LIN {X 0,Y 573.904,Z 122.065,A -85,B 0,C 180,E1 -2263.779,E2 -2263.779} C_VEL
LIN {X 0,Y 573.412,Z 118.44,A -85,B 0,C 180,E1 -2263.85,E2 -2263.85} C_VEL
LIN {X 0,Y 573.598,Z 96.264,A -85,B 0,C 180,E1 -2266.868,E2 -2266.868} C_VEL
LIN {X 0,Y 573.791,Z 74.375,A -85,B 0,C 180,E1 -2269.851,E2 -2269.851} C_VEL
LIN {X 0,Y 573.97,Z 52.577,A -85,B 0,C 180,E1 -2272.877,E2 -2272.877} C_VEL
LIN {X 0,Y 573.666,Z 48.09,A -85,B 0,C 180,E1 -2273.521,E2 -2273.521} C_VEL
LIN {X 0,Y 573.275,Z 46.079,A -85,B 0,C 180,E1 -2273.823,E2 -2273.823} C_VEL
LIN {X 0,Y 573.237,Z 46.08,A -85,B 0,C 180,E1 -2276.492,E2 -2276.492} C_VEL
LIN {X 0,Y 573.237,Z 46.078,A -85,B 0,C 180,E1 -2278.564,E2 -2278.564} C_VEL
LIN {X 0,Y 573.23,Z 46.075,A -85,B 0,C 180,E1 -2280.993,E2 -2280.993} C_VEL
LIN {X 0,Y 573.264,Z 46.076,A -85,B 0,C 180,E1 -2283.524,E2 -2283.524} C_VEL
LIN {X 0,Y 573.216,Z 46.083,A -85,B 0,C 180,E1 -2286.051,E2 -2286.051} C_VEL
LIN {X 0,Y 573.25,Z 46.073,A -85,B 0,C 180,E1 -2288.701,E2 -2288.701} C_VEL
LIN {X 0,Y 573.23,Z 46.085,A -85,B 0,C 180,E1 -2291.593,E2 -2291.593} C_VEL
LIN {X 0,Y 573.222,Z 46.077,A -85,B 0,C 180,E1 -2294.335,E2 -2294.335} C_VEL
LIN {X 0,Y 573.241,Z 46.083,A -85,B 0,C 180,E1 -2297.358,E2 -2297.358} C_VEL
LIN {X 0,Y 573.238,Z 46.075,A -85,B 0,C 180,E1 -2300.392,E2 -2300.392} C_VEL
LIN {X 0,Y 573.252,Z 46.08,A -85,B 0,C 180,E1 -2303.077,E2 -2303.077} C_VEL
LIN {X 0,Y 573.269,Z 46.073,A -85,B 0,C 180,E1 -2305.671,E2 -2305.671} C_VEL
LIN {X 0,Y 573.245,Z 46.074,A -85,B 0,C 180,E1 -2308.185,E2 -2308.185} C_VEL
LIN {X 0,Y 573.26,Z 46.076,A -85,B 0,C 180,E1 -2310.634,E2 -2310.634} C_VEL
LIN {X 0,Y 573.251,Z 46.081,A -85,B 0,C 180,E1 -2313.024,E2 -2313.024} C_VEL
LIN {X 0,Y 573.274,Z 46.073,A -85,B 0,C 180,E1 -2315.366,E2 -2315.366} C_VEL
LIN {X 0,Y 573.227,Z 46.08,A -85,B 0,C 180,E1 -2318.419,E2 -2318.419} C_VEL
LIN {X 0,Y 573.269,Z 46.08,A -85,B 0,C 180,E1 -2320.731,E2 -2320.731} C_VEL
LIN {X 0,Y 573.241,Z 46.074,A -85,B 0,C 180,E1 -2323.621,E2 -2323.621} C_VEL
LIN {X 0,Y 573.226,Z 46.086,A -85,B 0,C 180,E1 -2326.529,E2 -2326.529} C_VEL
LIN {X 0,Y 573.263,Z 46.076,A -85,B 0,C 180,E1 -2328.745,E2 -2328.745} C_VEL
LIN {X 0,Y 573.281,Z 46.069,A -85,B 0,C 180,E1 -2331.541,E2 -2331.541} C_VEL
LIN {X 0,Y 573.246,Z 46.075,A -85,B 0,C 180,E1 -2333.665,E2 -2333.665} C_VEL
LIN {X 0,Y 573.229,Z 46.079,A -85,B 0,C 180,E1 -2335.782,E2 -2335.782} C_VEL
LIN {X 0,Y 573.312,Z 46.071,A -85,B 0,C 180,E1 -2337.893,E2 -2337.893} C_VEL
LIN {X 0,Y 573.32,Z 46.066,A -85,B 0,C 180,E1 -2340.703,E2 -2340.703} C_VEL
LIN {X 0,Y 573.294,Z 46.068,A -85,B 0,C 180,E1 -2342.811,E2 -2342.811} C_VEL
LIN {X 0,Y 573.29,Z 46.073,A -85,B 0,C 180,E1 -2345.628,E2 -2345.628} C_VEL
LIN {X 0,Y 573.253,Z 46.074,A -85,B 0,C 180,E1 -2348.46,E2 -2348.46} C_VEL
LIN {X 0,Y 573.273,Z 46.074,A -85,B 0,C 180,E1 -2351.312,E2 -2351.312} C_VEL
LIN {X 0,Y 573.263,Z 46.072,A -85,B 0,C 180,E1 -2354.417,E2 -2354.417} C_VEL
LIN {X 0,Y 573.249,Z 46.076,A -85,B 0,C 180,E1 -2357.112,E2 -2357.112} C_VEL
LIN {X 0,Y 573.237,Z 46.076,A -85,B 0,C 180,E1 -2360.077,E2 -2360.077} C_VEL
LIN {X 0,Y 573.224,Z 46.076,A -85,B 0,C 180,E1 -2362.339,E2 -2362.339} C_VEL
LIN {X 0,Y 573.201,Z 46.079,A -85,B 0,C 180,E1 -2364.361,E2 -2364.361} C_VEL
LIN {X 0,Y 572.564,Z 46.164,A -85,B 0,C 180,E1 -2364.947,E2 -2364.947} C_VEL
LIN {X 0,Y 569.745,Z 46.52,A -85,B 0,C 180,E1 -2365.899,E2 -2365.899} C_VEL
LIN {X 0,Y 567.34,Z 46.822,A -85,B 0,C 180,E1 -2366.665,E2 -2366.665} C_VEL
LIN {X 0,Y 566.291,Z 46.949,A -85,B 0,C 180,E1 -2367.257,E2 -2367.257} C_VEL
LIN {X 0,Y 566.198,Z 46.957,A -85,B 0,C 180,E1 -2367.457,E2 -2367.457} C_VEL
LIN {X 0,Y 566.196,Z 46.953,A -85,B 0,C 180,E1 -2369.77,E2 -2369.77} C_VEL
LIN {X 0,Y 566.202,Z 46.952,A -85,B 0,C 180,E1 -2372.43,E2 -2372.43} C_VEL
LIN {X 0,Y 566.179,Z 46.964,A -85,B 0,C 180,E1 -2374.989,E2 -2374.989} C_VEL
LIN {X 0,Y 566.196,Z 46.954,A -85,B 0,C 180,E1 -2377.461,E2 -2377.461} C_VEL
LIN {X 0,Y 566.207,Z 46.952,A -85,B 0,C 180,E1 -2380.2,E2 -2380.2} C_VEL
LIN {X 0,Y 566.189,Z 46.957,A -85,B 0,C 180,E1 -2383.056,E2 -2383.056} C_VEL
LIN {X 0,Y 566.194,Z 46.954,A -85,B 0,C 180,E1 -2386.05,E2 -2386.05} C_VEL
LIN {X 0,Y 566.204,Z 46.952,A -85,B 0,C 180,E1 -2389.215,E2 -2389.215} C_VEL
LIN {X 0,Y 566.178,Z 46.954,A -85,B 0,C 180,E1 -2391.636,E2 -2391.636} C_VEL
LIN {X 0,Y 566.145,Z 46.967,A -85,B 0,C 180,E1 -2394.307,E2 -2394.307} C_VEL
LIN {X 0,Y 566.212,Z 46.951,A -85,B 0,C 180,E1 -2396.898,E2 -2396.898} C_VEL
LIN {X 0,Y 566.18,Z 46.954,A -85,B 0,C 180,E1 -2399.407,E2 -2399.407} C_VEL
LIN {X 0,Y 566.191,Z 46.958,A -85,B 0,C 180,E1 -2401.856,E2 -2401.856} C_VEL
LIN {X 0,Y 566.188,Z 46.959,A -85,B 0,C 180,E1 -2404.25,E2 -2404.25} C_VEL
LIN {X 0,Y 566.17,Z 46.956,A -85,B 0,C 180,E1 -2406.72,E2 -2406.72} C_VEL
LIN {X 0,Y 566.207,Z 46.956,A -85,B 0,C 180,E1 -2409.663,E2 -2409.663} C_VEL
LIN {X 0,Y 566.175,Z 46.964,A -85,B 0,C 180,E1 -2411.921,E2 -2411.921} C_VEL
LIN {X 0,Y 566.194,Z 46.954,A -85,B 0,C 180,E1 -2414.891,E2 -2414.891} C_VEL
LIN {X 0,Y 566.233,Z 46.954,A -85,B 0,C 180,E1 -2418.183,E2 -2418.183} C_VEL
LIN {X 0,Y 566.243,Z 47.146,A -85,B 0,C 180,E1 -2418.546,E2 -2418.546} C_VEL
LIN {X 0,Y 566.429,Z 52.827,A -85,B 0,C 180,E1 -2419.636,E2 -2419.636} C_VEL
LIN {X 0,Y 566.254,Z 68.023,A -85,B 0,C 180,E1 -2422.512,E2 -2422.512} C_VEL
LIN {X 0,Y 566.247,Z 70.905,A -85,B 0,C 180,E1 -2423.058,E2 -2423.058} C_VEL
LIN {X 0,Y 567.171,Z 77.845,A -85,B 0,C 180,E1 -2423.171,E2 -2423.171} C_VEL
LIN {X 0,Y 566.914,Z 176.791,A -85,B 0,C 180,E1 -2424.442,E2 -2424.442} C_VEL
LIN {X 0,Y 566.831,Z 189.95,A -85,B 0,C 180,E1 -2424.754,E2 -2424.754} C_VEL
LIN {X 0,Y 566.741,Z 202.54,A -85,B 0,C 180,E1 -2425.199,E2 -2425.199} C_VEL
LIN {X 0,Y 566.658,Z 213.764,A -85,B 0,C 180,E1 -2425.733,E2 -2425.733} C_VEL
LIN {X 0,Y 566.475,Z 225.38,A -85,B 0,C 180,E1 -2426.444,E2 -2426.444} C_VEL
LIN {X 0,Y 566.328,Z 235.815,A -85,B 0,C 180,E1 -2427.244,E2 -2427.244} C_VEL
LIN {X 0,Y 566.197,Z 246.089,A -85,B 0,C 180,E1 -2428.222,E2 -2428.222} C_VEL
LIN {X 0,Y 566.095,Z 255.035,A -85,B 0,C 180,E1 -2429.289,E2 -2429.289} C_VEL
LIN {X 0,Y 566.04,Z 262.266,A -85,B 0,C 180,E1 -2430.356,E2 -2430.356} C_VEL
LIN {X 0,Y 565.903,Z 268.085,A -85,B 0,C 180,E1 -2431.423,E2 -2431.423} C_VEL
LIN {X 0,Y 565.951,Z 272.675,A -85,B 0,C 180,E1 -2432.491,E2 -2432.491} C_VEL
LIN {X 0,Y 565.918,Z 276.184,A -85,B 0,C 180,E1 -2433.56,E2 -2433.56} C_VEL
LIN {X 0,Y 565.912,Z 277.971,A -85,B 0,C 180,E1 -2434.273,E2 -2434.273} C_VEL
LIN {X 0,Y 565.898,Z 280.275,A -85,B 0,C 180,E1 -2435.702,E2 -2435.702} C_VEL
LIN {X 0,Y 565.921,Z 280.892,A -85,B 0,C 180,E1 -2436.534,E2 -2436.534} C_VEL
LIN {X 0,Y 565.879,Z 280.721,A -85,B 0,C 180,E1 -2437.852,E2 -2437.852} C_VEL
LIN {X 0,Y 565.834,Z 279.017,A -85,B 0,C 180,E1 -2439.292,E2 -2439.292} C_VEL
LIN {X 0,Y 565.895,Z 277.513,A -85,B 0,C 180,E1 -2440.013,E2 -2440.013} C_VEL
LIN {X 0,Y 565.911,Z 274.239,A -85,B 0,C 180,E1 -2441.157,E2 -2441.157} C_VEL
LIN {X 0,Y 565.949,Z 270.275,A -85,B 0,C 180,E1 -2442.187,E2 -2442.187} C_VEL
LIN {X 0,Y 565.991,Z 263.857,A -85,B 0,C 180,E1 -2443.463,E2 -2443.463} C_VEL
LIN {X 0,Y 566.08,Z 257.636,A -85,B 0,C 180,E1 -2444.443,E2 -2444.443} C_VEL
LIN {X 0,Y 566.13,Z 249.591,A -85,B 0,C 180,E1 -2445.48,E2 -2445.48} C_VEL
LIN {X 0,Y 566.267,Z 239.776,A -85,B 0,C 180,E1 -2446.494,E2 -2446.494} C_VEL
LIN {X 0,Y 566.379,Z 229.838,A -85,B 0,C 180,E1 -2447.326,E2 -2447.326} C_VEL
LIN {X 0,Y 566.548,Z 218.884,A -85,B 0,C 180,E1 -2448.067,E2 -2448.067} C_VEL
LIN {X 0,Y 566.69,Z 206.505,A -85,B 0,C 180,E1 -2448.717,E2 -2448.717} C_VEL
LIN {X 0,Y 566.831,Z 193.521,A -85,B 0,C 180,E1 -2449.227,E2 -2449.227} C_VEL
LIN {X 0,Y 566.929,Z 180.647,A -85,B 0,C 180,E1 -2449.571,E2 -2449.571} C_VEL
LIN {X 0,Y 566.982,Z 162.278,A -85,B 0,C 180,E1 -2449.846,E2 -2449.846} C_VEL
LIN {X 0,Y 567.036,Z 75.255,A -85,B 0,C 180,E1 -2450.956,E2 -2450.956} C_VEL
LIN {X 0,Y 566.258,Z 70.809,A -85,B 0,C 180,E1 -2451.048,E2 -2451.048} C_VEL
LIN {X 0,Y 566.379,Z 56.348,A -85,B 0,C 180,E1 -2453.784,E2 -2453.784} C_VEL
LIN {X 0,Y 566.363,Z 48.024,A -85,B 0,C 180,E1 -2455.367,E2 -2455.367} C_VEL
LIN {X 0,Y 566.175,Z 46.961,A -85,B 0,C 180,E1 -2455.61,E2 -2455.61} C_VEL
LIN {X 0,Y 566.142,Z 46.967,A -85,B 0,C 180,E1 -2458.189,E2 -2458.189} C_VEL
LIN {X 0,Y 566.178,Z 46.955,A -85,B 0,C 180,E1 -2461.073,E2 -2461.073} C_VEL
LIN {X 0,Y 566.182,Z 46.958,A -85,B 0,C 180,E1 -2463.729,E2 -2463.729} C_VEL
LIN {X 0,Y 566.134,Z 46.962,A -85,B 0,C 180,E1 -2466.575,E2 -2466.575} C_VEL
LIN {X 0,Y 566.195,Z 46.954,A -85,B 0,C 180,E1 -2469.276,E2 -2469.276} C_VEL
LIN {X 0,Y 566.142,Z 46.965,A -85,B 0,C 180,E1 -2472.094,E2 -2472.094} C_VEL
LIN {X 0,Y 566.162,Z 46.954,A -85,B 0,C 180,E1 -2475.037,E2 -2475.037} C_VEL
LIN {X 0,Y 566.141,Z 46.964,A -85,B 0,C 180,E1 -2477.906,E2 -2477.906} C_VEL
LIN {X 0,Y 566.16,Z 46.957,A -85,B 0,C 180,E1 -2480.721,E2 -2480.721} C_VEL
LIN {X 0,Y 566.159,Z 46.961,A -85,B 0,C 180,E1 -2483.792,E2 -2483.792} C_VEL
LIN {X 0,Y 566.181,Z 46.954,A -85,B 0,C 180,E1 -2486.271,E2 -2486.271} C_VEL
LIN {X 0,Y 566.173,Z 46.958,A -85,B 0,C 180,E1 -2488.927,E2 -2488.927} C_VEL
LIN {X 0,Y 566.153,Z 46.958,A -85,B 0,C 180,E1 -2491.854,E2 -2491.854} C_VEL
LIN {X 0,Y 566.17,Z 46.955,A -85,B 0,C 180,E1 -2494.249,E2 -2494.249} C_VEL
LIN {X 0,Y 566.155,Z 46.96,A -85,B 0,C 180,E1 -2497.367,E2 -2497.367} C_VEL
LIN {X 0,Y 566.2,Z 46.952,A -85,B 0,C 180,E1 -2499.662,E2 -2499.662} C_VEL
LIN {X 0,Y 566.175,Z 46.954,A -85,B 0,C 180,E1 -2501.921,E2 -2501.921} C_VEL
LIN {X 0,Y 566.181,Z 46.955,A -85,B 0,C 180,E1 -2504.152,E2 -2504.152} C_VEL
LIN {X 0,Y 566.164,Z 46.961,A -85,B 0,C 180,E1 -2506.358,E2 -2506.358} C_VEL
LIN {X 0,Y 566.218,Z 46.95,A -85,B 0,C 180,E1 -2509.27,E2 -2509.27} C_VEL
LIN {X 0,Y 566.202,Z 46.956,A -85,B 0,C 180,E1 -2512.152,E2 -2512.152} C_VEL
LIN {X 0,Y 566.26,Z 46.945,A -85,B 0,C 180,E1 -2515.016,E2 -2515.016} C_VEL
LIN {X 0,Y 566.27,Z 46.947,A -85,B 0,C 180,E1 -2517.866,E2 -2517.866} C_VEL
LIN {X 0,Y 566.298,Z 46.94,A -85,B 0,C 180,E1 -2520.711,E2 -2520.711} C_VEL
LIN {X 0,Y 566.256,Z 46.945,A -85,B 0,C 180,E1 -2522.846,E2 -2522.846} C_VEL
LIN {X 0,Y 566.242,Z 46.95,A -85,B 0,C 180,E1 -2525.698,E2 -2525.698} C_VEL
LIN {X 0,Y 566.202,Z 46.952,A -85,B 0,C 180,E1 -2528.566,E2 -2528.566} C_VEL
LIN {X 0,Y 566.243,Z 46.95,A -85,B 0,C 180,E1 -2531.454,E2 -2531.454} C_VEL
LIN {X 0,Y 566.228,Z 46.948,A -85,B 0,C 180,E1 -2534.502,E2 -2534.502} C_VEL
LIN {X 0,Y 566.186,Z 46.958,A -85,B 0,C 180,E1 -2537.332,E2 -2537.332} C_VEL
LIN {X 0,Y 566.203,Z 46.959,A -85,B 0,C 180,E1 -2539.581,E2 -2539.581} C_VEL
LIN {X 0,Y 566.189,Z 46.954,A -85,B 0,C 180,E1 -2541.863,E2 -2541.863} C_VEL
LIN {X 0,Y 566.186,Z 46.959,A -85,B 0,C 180,E1 -2545.022,E2 -2545.022} C_VEL
LIN {X 0,Y 566.191,Z 46.96,A -85,B 0,C 180,E1 -2547.34,E2 -2547.34} C_VEL
LIN {X 0,Y 566.174,Z 46.956,A -85,B 0,C 180,E1 -2549.77,E2 -2549.77} C_VEL
LIN {X 0,Y 566.203,Z 46.953,A -85,B 0,C 180,E1 -2552.429,E2 -2552.429} C_VEL
LIN {X 0,Y 566.183,Z 46.959,A -85,B 0,C 180,E1 -2554.989,E2 -2554.989} C_VEL
LIN {X 0,Y 566.198,Z 46.952,A -85,B 0,C 180,E1 -2557.461,E2 -2557.461} C_VEL
LIN {X 0,Y 566.209,Z 46.953,A -85,B 0,C 180,E1 -2560.199,E2 -2560.199} C_VEL
LIN {X 0,Y 566.203,Z 46.955,A -85,B 0,C 180,E1 -2563.054,E2 -2563.054} C_VEL
LIN {X 0,Y 566.196,Z 46.954,A -85,B 0,C 180,E1 -2566.049,E2 -2566.049} C_VEL
LIN {X 0,Y 566.207,Z 46.951,A -85,B 0,C 180,E1 -2569.214,E2 -2569.214} C_VEL
LIN {X 0,Y 566.188,Z 46.954,A -85,B 0,C 180,E1 -2571.637,E2 -2571.637} C_VEL
LIN {X 0,Y 566.166,Z 46.963,A -85,B 0,C 180,E1 -2574.308,E2 -2574.308} C_VEL
LIN {X 0,Y 566.222,Z 46.951,A -85,B 0,C 180,E1 -2576.898,E2 -2576.898} C_VEL
LIN {X 0,Y 566.183,Z 46.956,A -85,B 0,C 180,E1 -2579.407,E2 -2579.407} C_VEL
LIN {X 0,Y 566.215,Z 46.959,A -85,B 0,C 180,E1 -2581.857,E2 -2581.857} C_VEL
LIN {X 0,Y 566.213,Z 46.955,A -85,B 0,C 180,E1 -2584.251,E2 -2584.251} C_VEL
LIN {X 0,Y 566.252,Z 47.124,A -85,B 0,C 180,E1 -2586.065,E2 -2586.065} C_VEL
LIN {X 0,Y 567,Z 52.241,A -85,B 0,C 180,E1 -2586.825,E2 -2586.825} C_VEL
LIN {X 0,Y 566.815,Z 68.49,A -85,B 0,C 180,E1 -2589.116,E2 -2589.116} C_VEL
LIN {X 0,Y 566.658,Z 86.112,A -85,B 0,C 180,E1 -2591.563,E2 -2591.563} C_VEL
LIN {X 0,Y 566.477,Z 106.389,A -85,B 0,C 180,E1 -2594.345,E2 -2594.345} C_VEL
LIN {X 0,Y 566.381,Z 118.444,A -85,B 0,C 180,E1 -2595.986,E2 -2595.986} C_VEL
LIN {X 0,Y 567.159,Z 125.165,A -85,B 0,C 180,E1 -2596.095,E2 -2596.095} C_VEL
LIN {X 0,Y 566.984,Z 226.934,A -85,B 0,C 180,E1 -2597.403,E2 -2597.403} C_VEL
LIN {X 0,Y 566.854,Z 240.208,A -85,B 0,C 180,E1 -2597.719,E2 -2597.719} C_VEL
LIN {X 0,Y 566.747,Z 252.371,A -85,B 0,C 180,E1 -2598.148,E2 -2598.148} C_VEL
LIN {X 0,Y 566.608,Z 264.187,A -85,B 0,C 180,E1 -2598.71,E2 -2598.71} C_VEL
LIN {X 0,Y 566.443,Z 276.19,A -85,B 0,C 180,E1 -2599.455,E2 -2599.455} C_VEL
LIN {X 0,Y 566.325,Z 286.603,A -85,B 0,C 180,E1 -2600.265,E2 -2600.265} C_VEL
LIN {X 0,Y 566.207,Z 295.111,A -85,B 0,C 180,E1 -2601.074,E2 -2601.074} C_VEL
LIN {X 0,Y 566.112,Z 302.959,A -85,B 0,C 180,E1 -2601.971,E2 -2601.971} C_VEL
LIN {X 0,Y 566.001,Z 310.621,A -85,B 0,C 180,E1 -2603.046,E2 -2603.046} C_VEL
LIN {X 0,Y 566.004,Z 317.678,A -85,B 0,C 180,E1 -2604.299,E2 -2604.299} C_VEL
LIN {X 0,Y 565.933,Z 322.372,A -85,B 0,C 180,E1 -2605.37,E2 -2605.37} C_VEL
LIN {X 0,Y 565.927,Z 325.958,A -85,B 0,C 180,E1 -2606.44,E2 -2606.44} C_VEL
LIN {X 0,Y 565.878,Z 327.807,A -85,B 0,C 180,E1 -2607.152,E2 -2607.152} C_VEL
LIN {X 0,Y 565.846,Z 330.183,A -85,B 0,C 180,E1 -2608.576,E2 -2608.576} C_VEL
LIN {X 0,Y 565.839,Z 331,A -85,B 0,C 180,E1 -2610,E2 -2610} C_VEL
LIN {X 0,Y 565.846,Z 330.185,A -85,B 0,C 180,E1 -2611.423,E2 -2611.423} C_VEL
LIN {X 0,Y 565.878,Z 327.81,A -85,B 0,C 180,E1 -2612.847,E2 -2612.847} C_VEL
LIN {X 0,Y 565.926,Z 324.896,A -85,B 0,C 180,E1 -2613.916,E2 -2613.916} C_VEL
LIN {X 0,Y 565.878,Z 320.949,A -85,B 0,C 180,E1 -2614.987,E2 -2614.987} C_VEL
LIN {X 0,Y 566.004,Z 315.868,A -85,B 0,C 180,E1 -2616.058,E2 -2616.058} C_VEL
LIN {X 0,Y 566.04,Z 309.468,A -85,B 0,C 180,E1 -2617.132,E2 -2617.132} C_VEL
LIN {X 0,Y 566.133,Z 301.479,A -85,B 0,C 180,E1 -2618.207,E2 -2618.207} C_VEL
LIN {X 0,Y 566.229,Z 293.335,A -85,B 0,C 180,E1 -2619.105,E2 -2619.105} C_VEL
LIN {X 0,Y 566.345,Z 283.4,A -85,B 0,C 180,E1 -2620.005,E2 -2620.005} C_VEL
LIN {X 0,Y 566.512,Z 272.292,A -85,B 0,C 180,E1 -2620.807,E2 -2620.807} C_VEL
LIN {X 0,Y 566.612,Z 261.175,A -85,B 0,C 180,E1 -2621.447,E2 -2621.447} C_VEL
LIN {X 0,Y 566.745,Z 248.981,A -85,B 0,C 180,E1 -2621.988,E2 -2621.988} C_VEL
LIN {X 0,Y 566.885,Z 236.181,A -85,B 0,C 180,E1 -2622.394,E2 -2622.394} C_VEL
LIN {X 0,Y 566.957,Z 222.612,A -85,B 0,C 180,E1 -2622.665,E2 -2622.665} C_VEL
LIN {X 0,Y 567.013,Z 122.67,A -85,B 0,C 180,E1 -2623.941,E2 -2623.941} C_VEL
LIN {X 0,Y 566.404,Z 118.364,A -85,B 0,C 180,E1 -2624.025,E2 -2624.025} C_VEL
LIN {X 0,Y 566.596,Z 95.699,A -85,B 0,C 180,E1 -2627.118,E2 -2627.118} C_VEL
LIN {X 0,Y 566.825,Z 73.929,A -85,B 0,C 180,E1 -2630.125,E2 -2630.125} C_VEL
LIN {X 0,Y 567.032,Z 53.651,A -85,B 0,C 180,E1 -2632.981,E2 -2632.981} C_VEL
LIN {X 0,Y 566.466,Z 48.214,A -85,B 0,C 180,E1 -2633.779,E2 -2633.779} C_VEL
LIN {X 0,Y 566.212,Z 46.959,A -85,B 0,C 180,E1 -2633.985,E2 -2633.985} C_VEL
LIN {X 0,Y 566.209,Z 46.954,A -85,B 0,C 180,E1 -2636.659,E2 -2636.659} C_VEL
LIN {X 0,Y 566.192,Z 46.953,A -85,B 0,C 180,E1 -2638.953,E2 -2638.953} C_VEL
LIN {X 0,Y 566.197,Z 46.954,A -85,B 0,C 180,E1 -2641.421,E2 -2641.421} C_VEL
LIN {X 0,Y 566.211,Z 46.958,A -85,B 0,C 180,E1 -2643.956,E2 -2643.956} C_VEL
LIN {X 0,Y 566.201,Z 46.952,A -85,B 0,C 180,E1 -2646.57,E2 -2646.57} C_VEL
LIN {X 0,Y 566.223,Z 46.958,A -85,B 0,C 180,E1 -2649.686,E2 -2649.686} C_VEL
LIN {X 0,Y 566.201,Z 46.952,A -85,B 0,C 180,E1 -2652.917,E2 -2652.917} C_VEL
LIN {X 0,Y 566.194,Z 46.954,A -85,B 0,C 180,E1 -2656.049,E2 -2656.049} C_VEL
LIN {X 0,Y 566.204,Z 46.958,A -85,B 0,C 180,E1 -2659.214,E2 -2659.214} C_VEL
LIN {X 0,Y 566.182,Z 46.958,A -85,B 0,C 180,E1 -2661.636,E2 -2661.636} C_VEL
LIN {X 0,Y 566.174,Z 46.955,A -85,B 0,C 180,E1 -2664.309,E2 -2664.309} C_VEL
LIN {X 0,Y 566.22,Z 46.955,A -85,B 0,C 180,E1 -2666.898,E2 -2666.898} C_VEL
LIN {X 0,Y 566.179,Z 46.958,A -85,B 0,C 180,E1 -2669.407,E2 -2669.407} C_VEL
LIN {X 0,Y 566.212,Z 46.95,A -85,B 0,C 180,E1 -2671.857,E2 -2671.857} C_VEL
LIN {X 0,Y 566.215,Z 46.951,A -85,B 0,C 180,E1 -2674.251,E2 -2674.251} C_VEL
LIN {X 0,Y 566.169,Z 46.963,A -85,B 0,C 180,E1 -2676.719,E2 -2676.719} C_VEL
LIN {X 0,Y 566.205,Z 46.951,A -85,B 0,C 180,E1 -2679.663,E2 -2679.663} C_VEL
LIN {X 0,Y 566.199,Z 46.961,A -85,B 0,C 180,E1 -2682.668,E2 -2682.668} C_VEL
LIN {X 0,Y 566.22,Z 46.949,A -85,B 0,C 180,E1 -2685.627,E2 -2685.627} C_VEL
LIN {X 0,Y 566.235,Z 46.953,A -85,B 0,C 180,E1 -2688.675,E2 -2688.675} C_VEL
LIN {X 0,Y 566.225,Z 46.948,A -85,B 0,C 180,E1 -2691.434,E2 -2691.434} C_VEL
LIN {X 0,Y 566.252,Z 46.954,A -85,B 0,C 180,E1 -2694.302,E2 -2694.302} C_VEL
LIN {X 0,Y 566.283,Z 46.946,A -85,B 0,C 180,E1 -2697.866,E2 -2697.866} C_VEL
LIN {X 0,Y 566.292,Z 46.941,A -85,B 0,C 180,E1 -2700.711,E2 -2700.711} C_VEL
LIN {X 0,Y 566.262,Z 46.944,A -85,B 0,C 180,E1 -2702.846,E2 -2702.846} C_VEL
LIN {X 0,Y 566.257,Z 46.95,A -85,B 0,C 180,E1 -2705.699,E2 -2705.699} C_VEL
LIN {X 0,Y 566.204,Z 46.951,A -85,B 0,C 180,E1 -2708.566,E2 -2708.566} C_VEL
LIN {X 0,Y 566.243,Z 46.951,A -85,B 0,C 180,E1 -2711.455,E2 -2711.455} C_VEL
LIN {X 0,Y 566.218,Z 46.949,A -85,B 0,C 180,E1 -2714.5,E2 -2714.5} C_VEL
LIN {X 0,Y 566.192,Z 46.958,A -85,B 0,C 180,E1 -2717.332,E2 -2717.332} C_VEL
LIN {X 0,Y 566.204,Z 46.951,A -85,B 0,C 180,E1 -2720.338,E2 -2720.338} C_VEL
LIN {X 0,Y 566.166,Z 46.964,A -85,B 0,C 180,E1 -2723.28,E2 -2723.28} C_VEL
LIN {X 0,Y 566.202,Z 46.954,A -85,B 0,C 180,E1 -2725.75,E2 -2725.75} C_VEL
LIN {X 0,Y 566.198,Z 46.957,A -85,B 0,C 180,E1 -2727.457,E2 -2727.457} C_VEL
LIN {X 0,Y 565.509,Z 47.04,A -85,B 0,C 180,E1 -2728.051,E2 -2728.051} C_VEL
LIN {X 0,Y 562.644,Z 47.401,A -85,B 0,C 180,E1 -2729.014,E2 -2729.014} C_VEL
LIN {X 0,Y 560.24,Z 47.696,A -85,B 0,C 180,E1 -2729.79,E2 -2729.79} C_VEL
LIN {X 0,Y 559.214,Z 47.822,A -85,B 0,C 180,E1 -2730.389,E2 -2730.389} C_VEL
LIN {X 0,Y 559.134,Z 47.834,A -85,B 0,C 180,E1 -2730.591,E2 -2730.591} C_VEL
LIN {X 0,Y 559.152,Z 47.834,A -85,B 0,C 180,E1 -2732.716,E2 -2732.716} C_VEL
LIN {X 0,Y 559.127,Z 47.837,A -85,B 0,C 180,E1 -2735.325,E2 -2735.325} C_VEL
LIN {X 0,Y 559.13,Z 47.832,A -85,B 0,C 180,E1 -2738.018,E2 -2738.018} C_VEL
LIN {X 0,Y 559.152,Z 47.839,A -85,B 0,C 180,E1 -2740.813,E2 -2740.813} C_VEL
LIN {X 0,Y 559.112,Z 47.834,A -85,B 0,C 180,E1 -2743.737,E2 -2743.737} C_VEL
LIN {X 0,Y 559.137,Z 47.835,A -85,B 0,C 180,E1 -2746.266,E2 -2746.266} C_VEL
LIN {X 0,Y 559.155,Z 47.83,A -85,B 0,C 180,E1 -2749.188,E2 -2749.188} C_VEL
LIN {X 0,Y 559.126,Z 47.835,A -85,B 0,C 180,E1 -2751.982,E2 -2751.982} C_VEL
LIN {X 0,Y 559.125,Z 47.836,A -85,B 0,C 180,E1 -2754.789,E2 -2754.789} C_VEL
LIN {X 0,Y 559.156,Z 47.829,A -85,B 0,C 180,E1 -2757.365,E2 -2757.365} C_VEL
LIN {X 0,Y 559.149,Z 47.839,A -85,B 0,C 180,E1 -2760.144,E2 -2760.144} C_VEL
LIN {X 0,Y 559.116,Z 47.834,A -85,B 0,C 180,E1 -2763.095,E2 -2763.095} C_VEL
LIN {X 0,Y 559.131,Z 47.834,A -85,B 0,C 180,E1 -2765.494,E2 -2765.494} C_VEL
LIN {X 0,Y 559.176,Z 47.827,A -85,B 0,C 180,E1 -2768.624,E2 -2768.624} C_VEL
LIN {X 0,Y 559.161,Z 47.828,A -85,B 0,C 180,E1 -2770.926,E2 -2770.926} C_VEL
LIN {X 0,Y 559.146,Z 47.838,A -85,B 0,C 180,E1 -2773.947,E2 -2773.947} C_VEL
LIN {X 0,Y 559.152,Z 47.834,A -85,B 0,C 180,E1 -2776.184,E2 -2776.184} C_VEL
LIN {X 0,Y 559.218,Z 47.985,A -85,B 0,C 180,E1 -2778.439,E2 -2778.439} C_VEL
LIN {X 0,Y 559.446,Z 53.482,A -85,B 0,C 180,E1 -2779.505,E2 -2779.505} C_VEL
LIN {X 0,Y 559.239,Z 66.852,A -85,B 0,C 180,E1 -2782.054,E2 -2782.054} C_VEL
LIN {X 0,Y 559.216,Z 71.137,A -85,B 0,C 180,E1 -2782.872,E2 -2782.872} C_VEL
LIN {X 0,Y 560.297,Z 78.121,A -85,B 0,C 180,E1 -2782.997,E2 -2782.997} C_VEL
LIN {X 0,Y 559.994,Z 177.044,A -85,B 0,C 180,E1 -2784.283,E2 -2784.283} C_VEL
LIN {X 0,Y 559.906,Z 190.225,A -85,B 0,C 180,E1 -2784.598,E2 -2784.598} C_VEL
LIN {X 0,Y 559.797,Z 202.829,A -85,B 0,C 180,E1 -2785.049,E2 -2785.049} C_VEL
LIN {X 0,Y 559.724,Z 214.048,A -85,B 0,C 180,E1 -2785.589,E2 -2785.589} C_VEL
LIN {X 0,Y 559.497,Z 225.628,A -85,B 0,C 180,E1 -2786.309,E2 -2786.309} C_VEL
LIN {X 0,Y 559.333,Z 236.012,A -85,B 0,C 180,E1 -2787.119,E2 -2787.119} C_VEL
LIN {X 0,Y 559.184,Z 245.396,A -85,B 0,C 180,E1 -2788.02,E2 -2788.02} C_VEL
LIN {X 0,Y 559.041,Z 254.451,A -85,B 0,C 180,E1 -2789.1,E2 -2789.1} C_VEL
LIN {X 0,Y 558.981,Z 261.743,A -85,B 0,C 180,E1 -2790.18,E2 -2790.18} C_VEL
LIN {X 0,Y 558.811,Z 268.513,A -85,B 0,C 180,E1 -2791.442,E2 -2791.442} C_VEL
LIN {X 0,Y 558.846,Z 273.007,A -85,B 0,C 180,E1 -2792.523,E2 -2792.523} C_VEL
LIN {X 0,Y 558.826,Z 276.438,A -85,B 0,C 180,E1 -2793.605,E2 -2793.605} C_VEL
LIN {X 0,Y 558.805,Z 278.151,A -85,B 0,C 180,E1 -2794.328,E2 -2794.328} C_VEL
LIN {X 0,Y 558.81,Z 280.373,A -85,B 0,C 180,E1 -2795.775,E2 -2795.775} C_VEL
LIN {X 0,Y 558.849,Z 280.894,A -85,B 0,C 180,E1 -2796.536,E2 -2796.536} C_VEL
LIN {X 0,Y 558.798,Z 280.661,A -85,B 0,C 180,E1 -2797.952,E2 -2797.952} C_VEL
LIN {X 0,Y 558.768,Z 279.965,A -85,B 0,C 180,E1 -2798.681,E2 -2798.681} C_VEL
LIN {X 0,Y 558.747,Z 278.853,A -85,B 0,C 180,E1 -2799.411,E2 -2799.411} C_VEL
LIN {X 0,Y 558.793,Z 277.287,A -85,B 0,C 180,E1 -2800.142,E2 -2800.142} C_VEL
LIN {X 0,Y 558.814,Z 274.3,A -85,B 0,C 180,E1 -2801.191,E2 -2801.191} C_VEL
LIN {X 0,Y 558.857,Z 269.867,A -85,B 0,C 180,E1 -2802.345,E2 -2802.345} C_VEL
LIN {X 0,Y 558.937,Z 263.371,A -85,B 0,C 180,E1 -2803.637,E2 -2803.637} C_VEL
LIN {X 0,Y 559.039,Z 256.239,A -85,B 0,C 180,E1 -2804.749,E2 -2804.749} C_VEL
LIN {X 0,Y 559.132,Z 247.254,A -85,B 0,C 180,E1 -2805.866,E2 -2805.866} C_VEL
LIN {X 0,Y 559.287,Z 237.983,A -85,B 0,C 180,E1 -2806.799,E2 -2806.799} C_VEL
LIN {X 0,Y 559.415,Z 227.589,A -85,B 0,C 180,E1 -2807.643,E2 -2807.643} C_VEL
LIN {X 0,Y 559.595,Z 215.958,A -85,B 0,C 180,E1 -2808.394,E2 -2808.394} C_VEL
LIN {X 0,Y 559.799,Z 203.75,A -85,B 0,C 180,E1 -2809.004,E2 -2809.004} C_VEL
LIN {X 0,Y 559.956,Z 191.238,A -85,B 0,C 180,E1 -2809.46,E2 -2809.46} C_VEL
LIN {X 0,Y 560.06,Z 178.166,A -85,B 0,C 180,E1 -2809.783,E2 -2809.783} C_VEL
LIN {X 0,Y 560.278,Z 89.454,A -85,B 0,C 180,E1 -2810.947,E2 -2810.947} C_VEL
LIN {X 0,Y 560.245,Z 76.666,A -85,B 0,C 180,E1 -2811.114,E2 -2811.114} C_VEL
LIN {X 0,Y 559.268,Z 71.081,A -85,B 0,C 180,E1 -2811.228,E2 -2811.228} C_VEL
LIN {X 0,Y 559.393,Z 56.026,A -85,B 0,C 180,E1 -2814.099,E2 -2814.099} C_VEL
LIN {X 0,Y 559.299,Z 48.823,A -85,B 0,C 180,E1 -2815.492,E2 -2815.492} C_VEL
LIN {X 0,Y 559.151,Z 47.837,A -85,B 0,C 180,E1 -2815.699,E2 -2815.699} C_VEL
LIN {X 0,Y 559.104,Z 47.844,A -85,B 0,C 180,E1 -2818.533,E2 -2818.533} C_VEL
LIN {X 0,Y 559.125,Z 47.834,A -85,B 0,C 180,E1 -2821.269,E2 -2821.269} C_VEL
LIN {X 0,Y 559.144,Z 47.838,A -85,B 0,C 180,E1 -2823.945,E2 -2823.945} C_VEL
LIN {X 0,Y 559.107,Z 47.835,A -85,B 0,C 180,E1 -2827.111,E2 -2827.111} C_VEL
LIN {X 0,Y 559.121,Z 47.842,A -85,B 0,C 180,E1 -2829.936,E2 -2829.936} C_VEL
LIN {X 0,Y 559.109,Z 47.835,A -85,B 0,C 180,E1 -2832.749,E2 -2832.749} C_VEL
LIN {X 0,Y 559.124,Z 47.84,A -85,B 0,C 180,E1 -2835.764,E2 -2835.764} C_VEL
LIN {X 0,Y 559.092,Z 47.838,A -85,B 0,C 180,E1 -2838.223,E2 -2838.223} C_VEL
LIN {X 0,Y 559.111,Z 47.837,A -85,B 0,C 180,E1 -2841.06,E2 -2841.06} C_VEL
LIN {X 0,Y 559.113,Z 47.838,A -85,B 0,C 180,E1 -2843.787,E2 -2843.787} C_VEL
LIN {X 0,Y 559.126,Z 47.833,A -85,B 0,C 180,E1 -2846.422,E2 -2846.422} C_VEL
LIN {X 0,Y 559.139,Z 47.835,A -85,B 0,C 180,E1 -2848.979,E2 -2848.979} C_VEL
LIN {X 0,Y 559.112,Z 47.837,A -85,B 0,C 180,E1 -2851.63,E2 -2851.63} C_VEL
LIN {X 0,Y 559.117,Z 47.834,A -85,B 0,C 180,E1 -2853.899,E2 -2853.899} C_VEL
LIN {X 0,Y 559.11,Z 47.842,A -85,B 0,C 180,E1 -2857.066,E2 -2857.066} C_VEL
LIN {X 0,Y 559.173,Z 47.83,A -85,B 0,C 180,E1 -2859.395,E2 -2859.395} C_VEL
LIN {X 0,Y 559.125,Z 47.832,A -85,B 0,C 180,E1 -2861.685,E2 -2861.685} C_VEL
LIN {X 0,Y 559.142,Z 47.831,A -85,B 0,C 180,E1 -2863.947,E2 -2863.947} C_VEL
LIN {X 0,Y 559.144,Z 47.833,A -85,B 0,C 180,E1 -2866.183,E2 -2866.183} C_VEL
LIN {X 0,Y 559.181,Z 47.827,A -85,B 0,C 180,E1 -2869.133,E2 -2869.133} C_VEL
LIN {X 0,Y 559.178,Z 47.83,A -85,B 0,C 180,E1 -2872.053,E2 -2872.053} C_VEL
LIN {X 0,Y 559.235,Z 47.82,A -85,B 0,C 180,E1 -2874.953,E2 -2874.953} C_VEL
LIN {X 0,Y 559.242,Z 47.822,A -85,B 0,C 180,E1 -2877.839,E2 -2877.839} C_VEL
LIN {X 0,Y 559.269,Z 47.816,A -85,B 0,C 180,E1 -2880.72,E2 -2880.72} C_VEL
LIN {X 0,Y 559.222,Z 47.821,A -85,B 0,C 180,E1 -2882.881,E2 -2882.881} C_VEL
LIN {X 0,Y 559.212,Z 47.827,A -85,B 0,C 180,E1 -2885.77,E2 -2885.77} C_VEL
LIN {X 0,Y 559.166,Z 47.828,A -85,B 0,C 180,E1 -2888.675,E2 -2888.675} C_VEL
LIN {X 0,Y 559.205,Z 47.828,A -85,B 0,C 180,E1 -2891.6,E2 -2891.6} C_VEL
LIN {X 0,Y 559.184,Z 47.825,A -85,B 0,C 180,E1 -2894.587,E2 -2894.587} C_VEL
LIN {X 0,Y 559.132,Z 47.839,A -85,B 0,C 180,E1 -2897.558,E2 -2897.558} C_VEL
LIN {X 0,Y 559.166,Z 47.832,A -85,B 0,C 180,E1 -2899.838,E2 -2899.838} C_VEL
LIN {X 0,Y 559.137,Z 47.83,A -85,B 0,C 180,E1 -2902.153,E2 -2902.153} C_VEL
LIN {X 0,Y 559.145,Z 47.838,A -85,B 0,C 180,E1 -2905.178,E2 -2905.178} C_VEL
LIN {X 0,Y 559.139,Z 47.833,A -85,B 0,C 180,E1 -2907.714,E2 -2907.714} C_VEL
LIN {X 0,Y 559.14,Z 47.831,A -85,B 0,C 180,E1 -2910.184,E2 -2910.184} C_VEL
LIN {X 0,Y 559.159,Z 47.833,A -85,B 0,C 180,E1 -2912.715,E2 -2912.715} C_VEL
LIN {X 0,Y 559.13,Z 47.832,A -85,B 0,C 180,E1 -2915.324,E2 -2915.324} C_VEL
LIN {X 0,Y 559.133,Z 47.831,A -85,B 0,C 180,E1 -2918.018,E2 -2918.018} C_VEL
LIN {X 0,Y 559.158,Z 47.837,A -85,B 0,C 180,E1 -2920.812,E2 -2920.812} C_VEL
LIN {X 0,Y 559.141,Z 47.831,A -85,B 0,C 180,E1 -2923.734,E2 -2923.734} C_VEL
LIN {X 0,Y 559.147,Z 47.835,A -85,B 0,C 180,E1 -2926.804,E2 -2926.804} C_VEL
LIN {X 0,Y 559.158,Z 47.829,A -85,B 0,C 180,E1 -2929.187,E2 -2929.187} C_VEL
LIN {X 0,Y 559.135,Z 47.836,A -85,B 0,C 180,E1 -2931.982,E2 -2931.982} C_VEL
LIN {X 0,Y 559.135,Z 47.834,A -85,B 0,C 180,E1 -2934.787,E2 -2934.787} C_VEL
LIN {X 0,Y 559.158,Z 47.831,A -85,B 0,C 180,E1 -2937.364,E2 -2937.364} C_VEL
LIN {X 0,Y 559.151,Z 47.839,A -85,B 0,C 180,E1 -2940.143,E2 -2940.143} C_VEL
LIN {X 0,Y 559.174,Z 47.829,A -85,B 0,C 180,E1 -2943.173,E2 -2943.173} C_VEL
LIN {X 0,Y 559.166,Z 47.838,A -85,B 0,C 180,E1 -2945.89,E2 -2945.89} C_VEL
LIN {X 0,Y 560.056,Z 53.466,A -85,B 0,C 180,E1 -2946.74,E2 -2946.74} C_VEL
LIN {X 0,Y 559.875,Z 68.194,A -85,B 0,C 180,E1 -2948.845,E2 -2948.845} C_VEL
LIN {X 0,Y 559.657,Z 87.155,A -85,B 0,C 180,E1 -2951.513,E2 -2951.513} C_VEL
LIN {X 0,Y 559.451,Z 107.432,A -85,B 0,C 180,E1 -2954.33,E2 -2954.33} C_VEL
LIN {X 0,Y 559.351,Z 118.042,A -85,B 0,C 180,E1 -2955.794,E2 -2955.794} C_VEL
LIN {X 0,Y 560.26,Z 125.885,A -85,B 0,C 180,E1 -2955.934,E2 -2955.934} C_VEL
LIN {X 0,Y 560.047,Z 226.675,A -85,B 0,C 180,E1 -2957.245,E2 -2957.245} C_VEL
LIN {X 0,Y 559.897,Z 239.981,A -85,B 0,C 180,E1 -2957.564,E2 -2957.564} C_VEL
LIN {X 0,Y 559.793,Z 252.184,A -85,B 0,C 180,E1 -2957.999,E2 -2957.999} C_VEL
LIN {X 0,Y 559.612,Z 263.724,A -85,B 0,C 180,E1 -2958.549,E2 -2958.549} C_VEL
LIN {X 0,Y 559.464,Z 274.813,A -85,B 0,C 180,E1 -2959.23,E2 -2959.23} C_VEL
LIN {X 0,Y 559.286,Z 285.509,A -85,B 0,C 180,E1 -2960.05,E2 -2960.05} C_VEL
LIN {X 0,Y 559.162,Z 295.111,A -85,B 0,C 180,E1 -2960.961,E2 -2960.961} C_VEL
LIN {X 0,Y 559.05,Z 302.959,A -85,B 0,C 180,E1 -2961.869,E2 -2961.869} C_VEL
LIN {X 0,Y 558.943,Z 310.621,A -85,B 0,C 180,E1 -2962.958,E2 -2962.958} C_VEL
LIN {X 0,Y 558.936,Z 317.678,A -85,B 0,C 180,E1 -2964.227,E2 -2964.227} C_VEL
LIN {X 0,Y 558.826,Z 322.372,A -85,B 0,C 180,E1 -2965.311,E2 -2965.311} C_VEL
LIN {X 0,Y 558.836,Z 325.957,A -85,B 0,C 180,E1 -2966.395,E2 -2966.395} C_VEL
LIN {X 0,Y 558.799,Z 327.806,A -85,B 0,C 180,E1 -2967.116,E2 -2967.116} C_VEL
LIN {X 0,Y 558.745,Z 330.182,A -85,B 0,C 180,E1 -2968.558,E2 -2968.558} C_VEL
LIN {X 0,Y 558.74,Z 331,A -85,B 0,C 180,E1 -2970,E2 -2970} C_VEL
LIN {X 0,Y 558.745,Z 330.184,A -85,B 0,C 180,E1 -2971.441,E2 -2971.441} C_VEL
LIN {X 0,Y 558.799,Z 327.81,A -85,B 0,C 180,E1 -2972.883,E2 -2972.883} C_VEL
LIN {X 0,Y 558.844,Z 324.896,A -85,B 0,C 180,E1 -2973.966,E2 -2973.966} C_VEL
LIN {X 0,Y 558.798,Z 320.949,A -85,B 0,C 180,E1 -2975.051,E2 -2975.051} C_VEL
LIN {X 0,Y 558.923,Z 315.868,A -85,B 0,C 180,E1 -2976.135,E2 -2976.135} C_VEL
LIN {X 0,Y 558.977,Z 309.468,A -85,B 0,C 180,E1 -2977.223,E2 -2977.223} C_VEL
LIN {X 0,Y 559.098,Z 301.479,A -85,B 0,C 180,E1 -2978.311,E2 -2978.311} C_VEL
LIN {X 0,Y 559.194,Z 293.334,A -85,B 0,C 180,E1 -2979.221,E2 -2979.221} C_VEL
LIN {X 0,Y 559.355,Z 283.365,A -85,B 0,C 180,E1 -2980.131,E2 -2980.131} C_VEL
LIN {X 0,Y 559.525,Z 272.304,A -85,B 0,C 180,E1 -2980.937,E2 -2980.937} C_VEL
LIN {X 0,Y 559.671,Z 260.31,A -85,B 0,C 180,E1 -2981.628,E2 -2981.628} C_VEL
LIN {X 0,Y 559.832,Z 247.574,A -85,B 0,C 180,E1 -2982.184,E2 -2982.184} C_VEL
LIN {X 0,Y 559.979,Z 234.115,A -85,B 0,C 180,E1 -2982.595,E2 -2982.595} C_VEL
LIN {X 0,Y 560.087,Z 220.833,A -85,B 0,C 180,E1 -2982.846,E2 -2982.846} C_VEL
LIN {X 0,Y 560.205,Z 123.963,A -85,B 0,C 180,E1 -2984.093,E2 -2984.093} C_VEL
LIN {X 0,Y 559.348,Z 118.057,A -85,B 0,C 180,E1 -2984.205,E2 -2984.205} C_VEL
LIN {X 0,Y 559.574,Z 96.192,A -85,B 0,C 180,E1 -2987.228,E2 -2987.228} C_VEL
LIN {X 0,Y 559.849,Z 74.99,A -85,B 0,C 180,E1 -2990.195,E2 -2990.195} C_VEL
LIN {X 0,Y 560.104,Z 54.797,A -85,B 0,C 180,E1 -2993.076,E2 -2993.076} C_VEL
LIN {X 0,Y 559.743,Z 50.65,A -85,B 0,C 180,E1 -2993.69,E2 -2993.69} C_VEL
LIN {X 0,Y 559.182,Z 47.835,A -85,B 0,C 180,E1 -2994.158,E2 -2994.158} C_VEL
LIN {X 0,Y 559.171,Z 47.829,A -85,B 0,C 180,E1 -2996.902,E2 -2996.902} C_VEL
LIN {X 0,Y 559.15,Z 47.838,A -85,B 0,C 180,E1 -2999.857,E2 -2999.857} C_VEL
LIN {X 0,Y 559.158,Z 47.829,A -85,B 0,C 180,E1 -3002.715,E2 -3002.715} C_VEL
LIN {X 0,Y 559.129,Z 47.835,A -85,B 0,C 180,E1 -3005.324,E2 -3005.324} C_VEL
LIN {X 0,Y 559.135,Z 47.836,A -85,B 0,C 180,E1 -3008.017,E2 -3008.017} C_VEL
LIN {X 0,Y 559.156,Z 47.829,A -85,B 0,C 180,E1 -3010.812,E2 -3010.812} C_VEL
LIN {X 0,Y 559.138,Z 47.838,A -85,B 0,C 180,E1 -3013.734,E2 -3013.734} C_VEL
LIN {X 0,Y 559.145,Z 47.831,A -85,B 0,C 180,E1 -3016.803,E2 -3016.803} C_VEL
LIN {X 0,Y 559.155,Z 47.835,A -85,B 0,C 180,E1 -3019.187,E2 -3019.187} C_VEL
LIN {X 0,Y 559.13,Z 47.833,A -85,B 0,C 180,E1 -3021.982,E2 -3021.982} C_VEL
LIN {X 0,Y 559.142,Z 47.834,A -85,B 0,C 180,E1 -3024.786,E2 -3024.786} C_VEL
LIN {X 0,Y 559.157,Z 47.834,A -85,B 0,C 180,E1 -3027.364,E2 -3027.364} C_VEL
LIN {X 0,Y 559.145,Z 47.83,A -85,B 0,C 180,E1 -3030.143,E2 -3030.143} C_VEL
LIN {X 0,Y 559.17,Z 47.834,A -85,B 0,C 180,E1 -3033.098,E2 -3033.098} C_VEL
LIN {X 0,Y 559.155,Z 47.83,A -85,B 0,C 180,E1 -3035.495,E2 -3035.495} C_VEL
LIN {X 0,Y 559.171,Z 47.834,A -85,B 0,C 180,E1 -3038.624,E2 -3038.624} C_VEL
LIN {X 0,Y 559.161,Z 47.834,A -85,B 0,C 180,E1 -3040.926,E2 -3040.926} C_VEL
LIN {X 0,Y 559.159,Z 47.83,A -85,B 0,C 180,E1 -3043.948,E2 -3043.948} C_VEL
LIN {X 0,Y 559.163,Z 47.832,A -85,B 0,C 180,E1 -3046.184,E2 -3046.184} C_VEL
LIN {X 0,Y 559.206,Z 47.83,A -85,B 0,C 180,E1 -3048.605,E2 -3048.605} C_VEL
LIN {X 0,Y 559.199,Z 47.828,A -85,B 0,C 180,E1 -3052.054,E2 -3052.054} C_VEL
LIN {X 0,Y 559.246,Z 47.818,A -85,B 0,C 180,E1 -3054.953,E2 -3054.953} C_VEL
LIN {X 0,Y 559.254,Z 47.821,A -85,B 0,C 180,E1 -3057.84,E2 -3057.84} C_VEL
LIN {X 0,Y 559.264,Z 47.817,A -85,B 0,C 180,E1 -3060.72,E2 -3060.72} C_VEL
LIN {X 0,Y 559.23,Z 47.82,A -85,B 0,C 180,E1 -3062.882,E2 -3062.882} C_VEL
LIN {X 0,Y 559.224,Z 47.828,A -85,B 0,C 180,E1 -3065.77,E2 -3065.77} C_VEL
LIN {X 0,Y 559.169,Z 47.827,A -85,B 0,C 180,E1 -3068.675,E2 -3068.675} C_VEL
LIN {X 0,Y 559.205,Z 47.83,A -85,B 0,C 180,E1 -3071.601,E2 -3071.601} C_VEL
LIN {X 0,Y 559.181,Z 47.826,A -85,B 0,C 180,E1 -3074.588,E2 -3074.588} C_VEL
LIN {X 0,Y 559.137,Z 47.841,A -85,B 0,C 180,E1 -3077.558,E2 -3077.558} C_VEL
LIN {X 0,Y 559.165,Z 47.832,A -85,B 0,C 180,E1 -3079.838,E2 -3079.838} C_VEL
LIN {X 0,Y 559.136,Z 47.832,A -85,B 0,C 180,E1 -3082.153,E2 -3082.153} C_VEL
LIN {X 0,Y 559.14,Z 47.839,A -85,B 0,C 180,E1 -3085.178,E2 -3085.178} C_VEL
LIN {X 0,Y 559.147,Z 47.832,A -85,B 0,C 180,E1 -3087.714,E2 -3087.714} C_VEL
LIN {X 0,Y 559.134,Z 47.834,A -85,B 0,C 180,E1 -3090.591,E2 -3090.591} C_VEL
LIN {X 0,Y 558.471,Z 47.922,A -85,B 0,C 180,E1 -3091.193,E2 -3091.193} C_VEL
LIN {X 0,Y 555.61,Z 48.279,A -85,B 0,C 180,E1 -3092.169,E2 -3092.169} C_VEL
LIN {X 0,Y 553.194,Z 48.579,A -85,B 0,C 180,E1 -3092.954,E2 -3092.954} C_VEL
LIN {X 0,Y 552.167,Z 48.702,A -85,B 0,C 180,E1 -3093.561,E2 -3093.561} C_VEL
LIN {X 0,Y 552.089,Z 48.71,A -85,B 0,C 180,E1 -3093.767,E2 -3093.767} C_VEL
LIN {X 0,Y 552.106,Z 48.714,A -85,B 0,C 180,E1 -3096.748,E2 -3096.748} C_VEL
LIN {X 0,Y 552.128,Z 48.705,A -85,B 0,C 180,E1 -3099.528,E2 -3099.528} C_VEL
LIN {X 0,Y 552.11,Z 48.711,A -85,B 0,C 180,E1 -3102.428,E2 -3102.428} C_VEL
LIN {X 0,Y 552.093,Z 48.709,A -85,B 0,C 180,E1 -3105.562,E2 -3105.562} C_VEL
LIN {X 0,Y 552.107,Z 48.714,A -85,B 0,C 180,E1 -3108.681,E2 -3108.681} C_VEL
LIN {X 0,Y 552.114,Z 48.706,A -85,B 0,C 180,E1 -3111.411,E2 -3111.411} C_VEL
LIN {X 0,Y 552.073,Z 48.717,A -85,B 0,C 180,E1 -3114.156,E2 -3114.156} C_VEL
LIN {X 0,Y 552.116,Z 48.708,A -85,B 0,C 180,E1 -3116.814,E2 -3116.814} C_VEL
LIN {X 0,Y 552.103,Z 48.708,A -85,B 0,C 180,E1 -3119.391,E2 -3119.391} C_VEL
LIN {X 0,Y 552.079,Z 48.716,A -85,B 0,C 180,E1 -3121.9,E2 -3121.9} C_VEL
LIN {X 0,Y 552.085,Z 48.711,A -85,B 0,C 180,E1 -3124.667,E2 -3124.667} C_VEL
LIN {X 0,Y 552.093,Z 48.712,A -85,B 0,C 180,E1 -3127.549,E2 -3127.549} C_VEL
LIN {X 0,Y 552.149,Z 48.704,A -85,B 0,C 180,E1 -3130.376,E2 -3130.376} C_VEL
LIN {X 0,Y 552.111,Z 48.707,A -85,B 0,C 180,E1 -3132.976,E2 -3132.976} C_VEL
LIN {X 0,Y 552.118,Z 48.713,A -85,B 0,C 180,E1 -3136.004,E2 -3136.004} C_VEL
LIN {X 0,Y 552.189,Z 48.799,A -85,B 0,C 180,E1 -3138.321,E2 -3138.321} C_VEL
LIN {X 0,Y 552.464,Z 54.147,A -85,B 0,C 180,E1 -3139.371,E2 -3139.371} C_VEL
LIN {X 0,Y 552.294,Z 65.663,A -85,B 0,C 180,E1 -3141.585,E2 -3141.585} C_VEL
LIN {X 0,Y 552.242,Z 71.663,A -85,B 0,C 180,E1 -3142.697,E2 -3142.697} C_VEL
LIN {X 0,Y 553.432,Z 79.69,A -85,B 0,C 180,E1 -3142.835,E2 -3142.835} C_VEL
LIN {X 0,Y 553.082,Z 178.428,A -85,B 0,C 180,E1 -3144.143,E2 -3144.143} C_VEL
LIN {X 0,Y 552.966,Z 191.999,A -85,B 0,C 180,E1 -3144.485,E2 -3144.485} C_VEL
LIN {X 0,Y 552.882,Z 204.202,A -85,B 0,C 180,E1 -3144.941,E2 -3144.941} C_VEL
LIN {X 0,Y 552.751,Z 215.923,A -85,B 0,C 180,E1 -3145.534,E2 -3145.534} C_VEL
LIN {X 0,Y 552.528,Z 227.192,A -85,B 0,C 180,E1 -3146.263,E2 -3146.263} C_VEL
LIN {X 0,Y 552.324,Z 237.367,A -85,B 0,C 180,E1 -3147.083,E2 -3147.083} C_VEL
LIN {X 0,Y 552.168,Z 246.537,A -85,B 0,C 180,E1 -3147.994,E2 -3147.994} C_VEL
LIN {X 0,Y 551.989,Z 255.429,A -85,B 0,C 180,E1 -3149.088,E2 -3149.088} C_VEL
LIN {X 0,Y 551.927,Z 262.605,A -85,B 0,C 180,E1 -3150.183,E2 -3150.183} C_VEL
LIN {X 0,Y 551.737,Z 269.211,A -85,B 0,C 180,E1 -3151.46,E2 -3151.46} C_VEL
LIN {X 0,Y 551.78,Z 273.571,A -85,B 0,C 180,E1 -3152.555,E2 -3152.555} C_VEL
LIN {X 0,Y 551.737,Z 276.891,A -85,B 0,C 180,E1 -3153.652,E2 -3153.652} C_VEL
LIN {X 0,Y 551.681,Z 279.799,A -85,B 0,C 180,E1 -3155.116,E2 -3155.116} C_VEL
LIN {X 0,Y 551.731,Z 281.073,A -85,B 0,C 180,E1 -3156.496,E2 -3156.496} C_VEL
LIN {X 0,Y 551.696,Z 281.135,A -85,B 0,C 180,E1 -3157.319,E2 -3157.319} C_VEL
LIN {X 0,Y 551.697,Z 280.792,A -85,B 0,C 180,E1 -3158.055,E2 -3158.055} C_VEL
LIN {X 0,Y 551.673,Z 280.062,A -85,B 0,C 180,E1 -3158.794,E2 -3158.794} C_VEL
LIN {X 0,Y 551.666,Z 278.884,A -85,B 0,C 180,E1 -3159.533,E2 -3159.533} C_VEL
LIN {X 0,Y 551.729,Z 276.346,A -85,B 0,C 180,E1 -3160.644,E2 -3160.644} C_VEL
LIN {X 0,Y 551.784,Z 272.777,A -85,B 0,C 180,E1 -3161.759,E2 -3161.759} C_VEL
LIN {X 0,Y 551.799,Z 268.06,A -85,B 0,C 180,E1 -3162.879,E2 -3162.879} C_VEL
LIN {X 0,Y 551.908,Z 262.045,A -85,B 0,C 180,E1 -3164.002,E2 -3164.002} C_VEL
LIN {X 0,Y 551.995,Z 254.501,A -85,B 0,C 180,E1 -3165.13,E2 -3165.13} C_VEL
LIN {X 0,Y 552.13,Z 246.754,A -85,B 0,C 180,E1 -3166.073,E2 -3166.073} C_VEL
LIN {X 0,Y 552.348,Z 237.263,A -85,B 0,C 180,E1 -3167.017,E2 -3167.017} C_VEL
LIN {X 0,Y 552.456,Z 226.598,A -85,B 0,C 180,E1 -3167.873,E2 -3167.873} C_VEL
LIN {X 0,Y 552.684,Z 214.665,A -85,B 0,C 180,E1 -3168.633,E2 -3168.633} C_VEL
LIN {X 0,Y 552.886,Z 202.935,A -85,B 0,C 180,E1 -3169.203,E2 -3169.203} C_VEL
LIN {X 0,Y 553.038,Z 189.783,A -85,B 0,C 180,E1 -3169.673,E2 -3169.673} C_VEL
LIN {X 0,Y 553.146,Z 176.539,A -85,B 0,C 180,E1 -3169.982,E2 -3169.982} C_VEL
LIN {X 0,Y 553.313,Z 76.962,A -85,B 0,C 180,E1 -3171.294,E2 -3171.294} C_VEL
LIN {X 0,Y 552.25,Z 71.351,A -85,B 0,C 180,E1 -3171.413,E2 -3171.413} C_VEL
LIN {X 0,Y 552.437,Z 55.711,A -85,B 0,C 180,E1 -3174.423,E2 -3174.423} C_VEL
LIN {X 0,Y 552.23,Z 49.476,A -85,B 0,C 180,E1 -3175.64,E2 -3175.64} C_VEL
LIN {X 0,Y 552.126,Z 48.712,A -85,B 0,C 180,E1 -3175.847,E2 -3175.847} C_VEL
LIN {X 0,Y 552.044,Z 48.718,A -85,B 0,C 180,E1 -3178.932,E2 -3178.932} C_VEL
LIN {X 0,Y 552.096,Z 48.71,A -85,B 0,C 180,E1 -3181.472,E2 -3181.472} C_VEL
LIN {X 0,Y 552.09,Z 48.718,A -85,B 0,C 180,E1 -3184.163,E2 -3184.163} C_VEL
LIN {X 0,Y 552.05,Z 48.715,A -85,B 0,C 180,E1 -3186.752,E2 -3186.752} C_VEL
LIN {X 0,Y 552.08,Z 48.714,A -85,B 0,C 180,E1 -3189.532,E2 -3189.532} C_VEL
LIN {X 0,Y 552.082,Z 48.713,A -85,B 0,C 180,E1 -3192.43,E2 -3192.43} C_VEL
LIN {X 0,Y 552.074,Z 48.714,A -85,B 0,C 180,E1 -3195.56,E2 -3195.56} C_VEL
LIN {X 0,Y 552.051,Z 48.714,A -85,B 0,C 180,E1 -3198.547,E2 -3198.547} C_VEL
LIN {X 0,Y 552.061,Z 48.72,A -85,B 0,C 180,E1 -3201.406,E2 -3201.406} C_VEL
LIN {X 0,Y 552.063,Z 48.712,A -85,B 0,C 180,E1 -3204.563,E2 -3204.563} C_VEL
LIN {X 0,Y 552.099,Z 48.715,A -85,B 0,C 180,E1 -3207.157,E2 -3207.157} C_VEL
LIN {X 0,Y 552.074,Z 48.712,A -85,B 0,C 180,E1 -3209.958,E2 -3209.958} C_VEL
LIN {X 0,Y 552.068,Z 48.714,A -85,B 0,C 180,E1 -3212.723,E2 -3212.723} C_VEL
LIN {X 0,Y 552.051,Z 48.722,A -85,B 0,C 180,E1 -3215.158,E2 -3215.158} C_VEL
LIN {X 0,Y 552.082,Z 48.711,A -85,B 0,C 180,E1 -3217.548,E2 -3217.548} C_VEL
LIN {X 0,Y 552.134,Z 48.706,A -85,B 0,C 180,E1 -3220.379,E2 -3220.379} C_VEL
LIN {X 0,Y 552.12,Z 48.711,A -85,B 0,C 180,E1 -3222.976,E2 -3222.976} C_VEL
LIN {X 0,Y 552.107,Z 48.708,A -85,B 0,C 180,E1 -3226.003,E2 -3226.003} C_VEL
LIN {X 0,Y 552.154,Z 48.704,A -85,B 0,C 180,E1 -3228.993,E2 -3228.993} C_VEL
LIN {X 0,Y 552.136,Z 48.706,A -85,B 0,C 180,E1 -3231.951,E2 -3231.951} C_VEL
LIN {X 0,Y 552.211,Z 48.696,A -85,B 0,C 180,E1 -3234.889,E2 -3234.889} C_VEL
LIN {X 0,Y 552.214,Z 48.697,A -85,B 0,C 180,E1 -3237.812,E2 -3237.812} C_VEL
LIN {X 0,Y 552.239,Z 48.691,A -85,B 0,C 180,E1 -3240.729,E2 -3240.729} C_VEL
LIN {X 0,Y 552.188,Z 48.697,A -85,B 0,C 180,E1 -3242.918,E2 -3242.918} C_VEL
LIN {X 0,Y 552.183,Z 48.704,A -85,B 0,C 180,E1 -3245.844,E2 -3245.844} C_VEL
LIN {X 0,Y 552.138,Z 48.703,A -85,B 0,C 180,E1 -3248.786,E2 -3248.786} C_VEL
LIN {X 0,Y 552.161,Z 48.707,A -85,B 0,C 180,E1 -3251.75,E2 -3251.75} C_VEL
LIN {X 0,Y 552.132,Z 48.704,A -85,B 0,C 180,E1 -3254.748,E2 -3254.748} C_VEL
LIN {X 0,Y 552.091,Z 48.714,A -85,B 0,C 180,E1 -3257.789,E2 -3257.789} C_VEL
LIN {X 0,Y 552.127,Z 48.706,A -85,B 0,C 180,E1 -3260.101,E2 -3260.101} C_VEL
LIN {X 0,Y 552.089,Z 48.707,A -85,B 0,C 180,E1 -3262.451,E2 -3262.451} C_VEL
LIN {X 0,Y 552.09,Z 48.717,A -85,B 0,C 180,E1 -3265.335,E2 -3265.335} C_VEL
LIN {X 0,Y 552.09,Z 48.709,A -85,B 0,C 180,E1 -3268.099,E2 -3268.099} C_VEL
LIN {X 0,Y 552.096,Z 48.711,A -85,B 0,C 180,E1 -3270.61,E2 -3270.61} C_VEL
LIN {X 0,Y 552.118,Z 48.712,A -85,B 0,C 180,E1 -3273.186,E2 -3273.186} C_VEL
LIN {X 0,Y 552.088,Z 48.706,A -85,B 0,C 180,E1 -3275.844,E2 -3275.844} C_VEL
LIN {X 0,Y 552.122,Z 48.711,A -85,B 0,C 180,E1 -3279.061,E2 -3279.061} C_VEL
LIN {X 0,Y 552.123,Z 48.706,A -85,B 0,C 180,E1 -3281.446,E2 -3281.446} C_VEL
LIN {X 0,Y 552.092,Z 48.718,A -85,B 0,C 180,E1 -3284.531,E2 -3284.531} C_VEL
LIN {X 0,Y 552.133,Z 48.704,A -85,B 0,C 180,E1 -3287.585,E2 -3287.585} C_VEL
LIN {X 0,Y 552.135,Z 48.712,A -85,B 0,C 180,E1 -3290.473,E2 -3290.473} C_VEL
LIN {X 0,Y 552.109,Z 48.707,A -85,B 0,C 180,E1 -3293.317,E2 -3293.317} C_VEL
LIN {X 0,Y 552.13,Z 48.71,A -85,B 0,C 180,E1 -3295.939,E2 -3295.939} C_VEL
LIN {X 0,Y 552.123,Z 48.71,A -85,B 0,C 180,E1 -3298.541,E2 -3298.541} C_VEL
LIN {X 0,Y 552.108,Z 48.711,A -85,B 0,C 180,E1 -3301.442,E2 -3301.442} C_VEL
LIN {X 0,Y 552.132,Z 48.708,A -85,B 0,C 180,E1 -3304.356,E2 -3304.356} C_VEL
LIN {X 0,Y 552.167,Z 48.892,A -85,B 0,C 180,E1 -3305.765,E2 -3305.765} C_VEL
LIN {X 0,Y 553.124,Z 55.716,A -85,B 0,C 180,E1 -3306.803,E2 -3306.803} C_VEL
LIN {X 0,Y 552.884,Z 70.602,A -85,B 0,C 180,E1 -3308.955,E2 -3308.955} C_VEL
LIN {X 0,Y 552.636,Z 89.551,A -85,B 0,C 180,E1 -3311.654,E2 -3311.654} C_VEL
LIN {X 0,Y 552.416,Z 108.45,A -85,B 0,C 180,E1 -3314.315,E2 -3314.315} C_VEL
LIN {X 0,Y 552.337,Z 117.82,A -85,B 0,C 180,E1 -3315.625,E2 -3315.625} C_VEL
LIN {X 0,Y 553.364,Z 126.039,A -85,B 0,C 180,E1 -3315.761,E2 -3315.761} C_VEL
LIN {X 0,Y 553.131,Z 226.336,A -85,B 0,C 180,E1 -3317.083,E2 -3317.083} C_VEL
LIN {X 0,Y 552.975,Z 239.646,A -85,B 0,C 180,E1 -3317.405,E2 -3317.405} C_VEL
LIN {X 0,Y 552.837,Z 251.843,A -85,B 0,C 180,E1 -3317.845,E2 -3317.845} C_VEL
LIN {X 0,Y 552.638,Z 263.393,A -85,B 0,C 180,E1 -3318.402,E2 -3318.402} C_VEL
LIN {X 0,Y 552.468,Z 274.483,A -85,B 0,C 180,E1 -3319.092,E2 -3319.092} C_VEL
LIN {X 0,Y 552.26,Z 285.18,A -85,B 0,C 180,E1 -3319.922,E2 -3319.922} C_VEL
LIN {X 0,Y 552.11,Z 294.823,A -85,B 0,C 180,E1 -3320.844,E2 -3320.844} C_VEL
LIN {X 0,Y 551.984,Z 302.729,A -85,B 0,C 180,E1 -3321.765,E2 -3321.765} C_VEL
LIN {X 0,Y 551.889,Z 310.453,A -85,B 0,C 180,E1 -3322.867,E2 -3322.867} C_VEL
LIN {X 0,Y 551.845,Z 317.575,A -85,B 0,C 180,E1 -3324.152,E2 -3324.152} C_VEL
LIN {X 0,Y 551.723,Z 322.309,A -85,B 0,C 180,E1 -3325.25,E2 -3325.25} C_VEL
LIN {X 0,Y 551.75,Z 325.931,A -85,B 0,C 180,E1 -3326.348,E2 -3326.348} C_VEL
LIN {X 0,Y 551.723,Z 327.795,A -85,B 0,C 180,E1 -3327.079,E2 -3327.079} C_VEL
LIN {X 0,Y 551.645,Z 330.179,A -85,B 0,C 180,E1 -3328.54,E2 -3328.54} C_VEL
LIN {X 0,Y 551.64,Z 331,A -85,B 0,C 180,E1 -3330,E2 -3330} C_VEL
LIN {X 0,Y 551.645,Z 330.182,A -85,B 0,C 180,E1 -3331.46,E2 -3331.46} C_VEL
LIN {X 0,Y 551.723,Z 327.799,A -85,B 0,C 180,E1 -3332.92,E2 -3332.92} C_VEL
LIN {X 0,Y 551.764,Z 324.86,A -85,B 0,C 180,E1 -3334.017,E2 -3334.017} C_VEL
LIN {X 0,Y 551.723,Z 320.872,A -85,B 0,C 180,E1 -3335.116,E2 -3335.116} C_VEL
LIN {X 0,Y 551.798,Z 315.057,A -85,B 0,C 180,E1 -3336.342,E2 -3336.342} C_VEL
LIN {X 0,Y 551.909,Z 308.052,A -85,B 0,C 180,E1 -3337.5,E2 -3337.5} C_VEL
LIN {X 0,Y 552.041,Z 299.747,A -85,B 0,C 180,E1 -3338.603,E2 -3338.603} C_VEL
LIN {X 0,Y 552.167,Z 291.235,A -85,B 0,C 180,E1 -3339.524,E2 -3339.524} C_VEL
LIN {X 0,Y 552.391,Z 280.723,A -85,B 0,C 180,E1 -3340.445,E2 -3340.445} C_VEL
LIN {X 0,Y 552.535,Z 269.859,A -85,B 0,C 180,E1 -3341.215,E2 -3341.215} C_VEL
LIN {X 0,Y 552.722,Z 258.929,A -85,B 0,C 180,E1 -3341.831,E2 -3341.831} C_VEL
LIN {X 0,Y 552.884,Z 247.245,A -85,B 0,C 180,E1 -3342.34,E2 -3342.34} C_VEL
LIN {X 0,Y 553.034,Z 233.786,A -85,B 0,C 180,E1 -3342.756,E2 -3342.756} C_VEL
LIN {X 0,Y 553.17,Z 220.497,A -85,B 0,C 180,E1 -3343.009,E2 -3343.009} C_VEL
LIN {X 0,Y 553.224,Z 124.104,A -85,B 0,C 180,E1 -3344.268,E2 -3344.268} C_VEL
LIN {X 0,Y 552.346,Z 117.718,A -85,B 0,C 180,E1 -3344.392,E2 -3344.392} C_VEL
LIN {X 0,Y 552.56,Z 97.423,A -85,B 0,C 180,E1 -3347.236,E2 -3347.236} C_VEL
LIN {X 0,Y 552.88,Z 76.065,A -85,B 0,C 180,E1 -3350.267,E2 -3350.267} C_VEL
LIN {X 0,Y 553.16,Z 55.791,A -85,B 0,C 180,E1 -3353.195,E2 -3353.195} C_VEL
LIN {X 0,Y 552.452,Z 50.342,A -85,B 0,C 180,E1 -3354.022,E2 -3354.022} C_VEL
LIN {X 0,Y 552.128,Z 48.713,A -85,B 0,C 180,E1 -3354.287,E2 -3354.287} C_VEL
LIN {X 0,Y 552.14,Z 48.705,A -85,B 0,C 180,E1 -3357.273,E2 -3357.273} C_VEL
LIN {X 0,Y 552.119,Z 48.715,A -85,B 0,C 180,E1 -3360.051,E2 -3360.051} C_VEL
LIN {X 0,Y 552.116,Z 48.706,A -85,B 0,C 180,E1 -3362.846,E2 -3362.846} C_VEL
LIN {X 0,Y 552.078,Z 48.714,A -85,B 0,C 180,E1 -3365.44,E2 -3365.44} C_VEL
LIN {X 0,Y 552.099,Z 48.715,A -85,B 0,C 180,E1 -3367.886,E2 -3367.886} C_VEL
LIN {X 0,Y 552.11,Z 48.707,A -85,B 0,C 180,E1 -3370.481,E2 -3370.481} C_VEL
LIN {X 0,Y 552.107,Z 48.714,A -85,B 0,C 180,E1 -3373.424,E2 -3373.424} C_VEL
LIN {X 0,Y 552.107,Z 48.707,A -85,B 0,C 180,E1 -3376.576,E2 -3376.576} C_VEL
LIN {X 0,Y 552.108,Z 48.714,A -85,B 0,C 180,E1 -3379.519,E2 -3379.519} C_VEL
LIN {X 0,Y 552.091,Z 48.709,A -85,B 0,C 180,E1 -3382.336,E2 -3382.336} C_VEL
LIN {X 0,Y 552.116,Z 48.713,A -85,B 0,C 180,E1 -3385.053,E2 -3385.053} C_VEL
LIN {X 0,Y 552.117,Z 48.707,A -85,B 0,C 180,E1 -3387.681,E2 -3387.681} C_VEL
LIN {X 0,Y 552.109,Z 48.707,A -85,B 0,C 180,E1 -3390.235,E2 -3390.235} C_VEL
LIN {X 0,Y 552.138,Z 48.712,A -85,B 0,C 180,E1 -3393,E2 -3393} C_VEL
LIN {X 0,Y 552.113,Z 48.711,A -85,B 0,C 180,E1 -3395.161,E2 -3395.161} C_VEL
LIN {X 0,Y 552.126,Z 48.708,A -85,B 0,C 180,E1 -3398.337,E2 -3398.337} C_VEL
LIN {X 0,Y 552.15,Z 48.711,A -85,B 0,C 180,E1 -3400.674,E2 -3400.674} C_VEL
LIN {X 0,Y 552.11,Z 48.707,A -85,B 0,C 180,E1 -3403.737,E2 -3403.737} C_VEL
LIN {X 0,Y 552.129,Z 48.706,A -85,B 0,C 180,E1 -3406.004,E2 -3406.004} C_VEL
LIN {X 0,Y 552.161,Z 48.702,A -85,B 0,C 180,E1 -3408.993,E2 -3408.993} C_VEL
LIN {X 0,Y 552.154,Z 48.705,A -85,B 0,C 180,E1 -3411.952,E2 -3411.952} C_VEL
LIN {X 0,Y 552.222,Z 48.694,A -85,B 0,C 180,E1 -3414.889,E2 -3414.889} C_VEL
LIN {X 0,Y 552.225,Z 48.696,A -85,B 0,C 180,E1 -3417.812,E2 -3417.812} C_VEL
LIN {X 0,Y 552.235,Z 48.692,A -85,B 0,C 180,E1 -3420.729,E2 -3420.729} C_VEL
LIN {X 0,Y 552.198,Z 48.696,A -85,B 0,C 180,E1 -3422.918,E2 -3422.918} C_VEL
LIN {X 0,Y 552.193,Z 48.705,A -85,B 0,C 180,E1 -3425.844,E2 -3425.844} C_VEL
LIN {X 0,Y 552.141,Z 48.703,A -85,B 0,C 180,E1 -3428.786,E2 -3428.786} C_VEL
LIN {X 0,Y 552.162,Z 48.709,A -85,B 0,C 180,E1 -3431.751,E2 -3431.751} C_VEL
LIN {X 0,Y 552.129,Z 48.704,A -85,B 0,C 180,E1 -3434.749,E2 -3434.749} C_VEL
LIN {X 0,Y 552.095,Z 48.714,A -85,B 0,C 180,E1 -3437.789,E2 -3437.789} C_VEL
LIN {X 0,Y 552.126,Z 48.706,A -85,B 0,C 180,E1 -3440.102,E2 -3440.102} C_VEL
LIN {X 0,Y 552.087,Z 48.709,A -85,B 0,C 180,E1 -3442.451,E2 -3442.451} C_VEL
LIN {X 0,Y 552.109,Z 48.711,A -85,B 0,C 180,E1 -3445.646,E2 -3445.646} C_VEL
LIN {X 0,Y 552.093,Z 48.709,A -85,B 0,C 180,E1 -3448.1,E2 -3448.1} C_VEL
LIN {X 0,Y 552.098,Z 48.71,A -85,B 0,C 180,E1 -3450.61,E2 -3450.61} C_VEL
LIN {X 0,Y 552.106,Z 48.714,A -85,B 0,C 180,E1 -3453.187,E2 -3453.187} C_VEL
LIN {X 0,Y 552.089,Z 48.71,A -85,B 0,C 180,E1 -3453.767,E2 -3453.767} C_VEL
LIN {X 0,Y 551.448,Z 48.791,A -85,B 0,C 180,E1 -3454.375,E2 -3454.375} C_VEL
LIN {X 0,Y 548.637,Z 49.15,A -85,B 0,C 180,E1 -3455.364,E2 -3455.364} C_VEL
LIN {X 0,Y 546.231,Z 49.455,A -85,B 0,C 180,E1 -3456.159,E2 -3456.159} C_VEL
LIN {X 0,Y 545.167,Z 49.583,A -85,B 0,C 180,E1 -3456.773,E2 -3456.773} C_VEL
LIN {X 0,Y 545.064,Z 49.593,A -85,B 0,C 180,E1 -3456.981,E2 -3456.981} C_VEL
LIN {X 0,Y 545.064,Z 49.585,A -85,B 0,C 180,E1 -3460.143,E2 -3460.143} C_VEL
LIN {X 0,Y 545.024,Z 49.593,A -85,B 0,C 180,E1 -3463.113,E2 -3463.113} C_VEL
LIN {X 0,Y 545.051,Z 49.589,A -85,B 0,C 180,E1 -3466.227,E2 -3466.227} C_VEL
LIN {X 0,Y 545.072,Z 49.588,A -85,B 0,C 180,E1 -3468.885,E2 -3468.885} C_VEL
LIN {X 0,Y 545.079,Z 49.587,A -85,B 0,C 180,E1 -3470.818,E2 -3470.818} C_VEL
LIN {X 0,Y 545.033,Z 49.589,A -85,B 0,C 180,E1 -3473.619,E2 -3473.619} C_VEL
LIN {X 0,Y 545.066,Z 49.593,A -85,B 0,C 180,E1 -3476.328,E2 -3476.328} C_VEL
LIN {X 0,Y 545.069,Z 49.584,A -85,B 0,C 180,E1 -3478.953,E2 -3478.953} C_VEL
LIN {X 0,Y 545.078,Z 49.584,A -85,B 0,C 180,E1 -3481.507,E2 -3481.507} C_VEL
LIN {X 0,Y 545.036,Z 49.591,A -85,B 0,C 180,E1 -3484.506,E2 -3484.506} C_VEL
LIN {X 0,Y 545.038,Z 49.588,A -85,B 0,C 180,E1 -3487.242,E2 -3487.242} C_VEL
LIN {X 0,Y 545.12,Z 49.579,A -85,B 0,C 180,E1 -3490.415,E2 -3490.415} C_VEL
LIN {X 0,Y 545.043,Z 49.592,A -85,B 0,C 180,E1 -3493.52,E2 -3493.52} C_VEL
LIN {X 0,Y 545.083,Z 49.591,A -85,B 0,C 180,E1 -3495.82,E2 -3495.82} C_VEL
LIN {X 0,Y 545.147,Z 49.715,A -85,B 0,C 180,E1 -3498.22,E2 -3498.22} C_VEL
LIN {X 0,Y 545.483,Z 54.823,A -85,B 0,C 180,E1 -3499.233,E2 -3499.233} C_VEL
LIN {X 0,Y 545.314,Z 66.388,A -85,B 0,C 180,E1 -3501.477,E2 -3501.477} C_VEL
LIN {X 0,Y 545.229,Z 71.656,A -85,B 0,C 180,E1 -3502.493,E2 -3502.493} C_VEL
LIN {X 0,Y 546.567,Z 80.208,A -85,B 0,C 180,E1 -3502.655,E2 -3502.655} C_VEL
LIN {X 0,Y 546.18,Z 178.68,A -85,B 0,C 180,E1 -3503.976,E2 -3503.976} C_VEL
LIN {X 0,Y 546.047,Z 192.275,A -85,B 0,C 180,E1 -3504.322,E2 -3504.322} C_VEL
LIN {X 0,Y 545.957,Z 204.487,A -85,B 0,C 180,E1 -3504.784,E2 -3504.784} C_VEL
LIN {X 0,Y 545.805,Z 216.218,A -85,B 0,C 180,E1 -3505.384,E2 -3505.384} C_VEL
LIN {X 0,Y 545.559,Z 227.492,A -85,B 0,C 180,E1 -3506.122,E2 -3506.122} C_VEL
LIN {X 0,Y 545.338,Z 237.67,A -85,B 0,C 180,E1 -3506.953,E2 -3506.953} C_VEL
LIN {X 0,Y 545.187,Z 246.005,A -85,B 0,C 180,E1 -3507.784,E2 -3507.784} C_VEL
LIN {X 0,Y 544.959,Z 255.074,A -85,B 0,C 180,E1 -3508.892,E2 -3508.892} C_VEL
LIN {X 0,Y 544.884,Z 262.367,A -85,B 0,C 180,E1 -3510,E2 -3510} C_VEL
LIN {X 0,Y 544.739,Z 268.246,A -85,B 0,C 180,E1 -3511.109,E2 -3511.109} C_VEL
LIN {X 0,Y 544.644,Z 272.901,A -85,B 0,C 180,E1 -3512.219,E2 -3512.219} C_VEL
LIN {X 0,Y 544.686,Z 276.462,A -85,B 0,C 180,E1 -3513.329,E2 -3513.329} C_VEL
LIN {X 0,Y 544.61,Z 279.041,A -85,B 0,C 180,E1 -3514.441,E2 -3514.441} C_VEL
LIN {X 0,Y 544.602,Z 280.256,A -85,B 0,C 180,E1 -3515.183,E2 -3515.183} C_VEL
LIN {X 0,Y 544.668,Z 281.396,A -85,B 0,C 180,E1 -3516.506,E2 -3516.506} C_VEL
LIN {X 0,Y 544.608,Z 281.435,A -85,B 0,C 180,E1 -3517.415,E2 -3517.415} C_VEL
LIN {X 0,Y 544.613,Z 281.054,A -85,B 0,C 180,E1 -3518.161,E2 -3518.161} C_VEL
LIN {X 0,Y 544.591,Z 280.254,A -85,B 0,C 180,E1 -3518.909,E2 -3518.909} C_VEL
LIN {X 0,Y 544.592,Z 279.025,A -85,B 0,C 180,E1 -3519.658,E2 -3519.658} C_VEL
LIN {X 0,Y 544.661,Z 276.403,A -85,B 0,C 180,E1 -3520.784,E2 -3520.784} C_VEL
LIN {X 0,Y 544.708,Z 272.743,A -85,B 0,C 180,E1 -3521.914,E2 -3521.914} C_VEL
LIN {X 0,Y 544.758,Z 267.929,A -85,B 0,C 180,E1 -3523.048,E2 -3523.048} C_VEL
LIN {X 0,Y 544.873,Z 261.806,A -85,B 0,C 180,E1 -3524.186,E2 -3524.186} C_VEL
LIN {X 0,Y 544.984,Z 254.14,A -85,B 0,C 180,E1 -3525.329,E2 -3525.329} C_VEL
LIN {X 0,Y 545.159,Z 246.235,A -85,B 0,C 180,E1 -3526.284,E2 -3526.284} C_VEL
LIN {X 0,Y 545.346,Z 236.498,A -85,B 0,C 180,E1 -3527.242,E2 -3527.242} C_VEL
LIN {X 0,Y 545.562,Z 225.616,A -85,B 0,C 180,E1 -3528.107,E2 -3528.107} C_VEL
LIN {X 0,Y 545.745,Z 215.001,A -85,B 0,C 180,E1 -3528.781,E2 -3528.781} C_VEL
LIN {X 0,Y 545.953,Z 203.274,A -85,B 0,C 180,E1 -3529.359,E2 -3529.359} C_VEL
LIN {X 0,Y 546.132,Z 189.781,A -85,B 0,C 180,E1 -3529.845,E2 -3529.845} C_VEL
LIN {X 0,Y 546.248,Z 176.673,A -85,B 0,C 180,E1 -3530.151,E2 -3530.151} C_VEL
LIN {X 0,Y 546.433,Z 77.858,A -85,B 0,C 180,E1 -3531.47,E2 -3531.47} C_VEL
LIN {X 0,Y 545.276,Z 71.657,A -85,B 0,C 180,E1 -3531.598,E2 -3531.598} C_VEL
LIN {X 0,Y 545.47,Z 56.44,A -85,B 0,C 180,E1 -3534.552,E2 -3534.552} C_VEL
LIN {X 0,Y 545.228,Z 50.421,A -85,B 0,C 180,E1 -3535.733,E2 -3535.733} C_VEL
LIN {X 0,Y 545.08,Z 49.59,A -85,B 0,C 180,E1 -3535.936,E2 -3535.936} C_VEL
LIN {X 0,Y 545.02,Z 49.592,A -85,B 0,C 180,E1 -3539.341,E2 -3539.341} C_VEL
LIN {X 0,Y 545.044,Z 49.592,A -85,B 0,C 180,E1 -3541.916,E2 -3541.916} C_VEL
LIN {X 0,Y 545.044,Z 49.591,A -85,B 0,C 180,E1 -3544.566,E2 -3544.566} C_VEL
LIN {X 0,Y 545.009,Z 49.592,A -85,B 0,C 180,E1 -3547.307,E2 -3547.307} C_VEL
LIN {X 0,Y 545.009,Z 49.598,A -85,B 0,C 180,E1 -3550.148,E2 -3550.148} C_VEL
LIN {X 0,Y 545.001,Z 49.594,A -85,B 0,C 180,E1 -3553.115,E2 -3553.115} C_VEL
LIN {X 0,Y 545.031,Z 49.596,A -85,B 0,C 180,E1 -3555.868,E2 -3555.868} C_VEL
LIN {X 0,Y 544.994,Z 49.593,A -85,B 0,C 180,E1 -3558.877,E2 -3558.877} C_VEL
LIN {X 0,Y 545.006,Z 49.596,A -85,B 0,C 180,E1 -3561.87,E2 -3561.87} C_VEL
LIN {X 0,Y 545.023,Z 49.589,A -85,B 0,C 180,E1 -3564.53,E2 -3564.53} C_VEL
LIN {X 0,Y 545.054,Z 49.593,A -85,B 0,C 180,E1 -3567.21,E2 -3567.21} C_VEL
LIN {X 0,Y 545.023,Z 49.592,A -85,B 0,C 180,E1 -3569.808,E2 -3569.808} C_VEL
LIN {X 0,Y 545.004,Z 49.591,A -85,B 0,C 180,E1 -3572.339,E2 -3572.339} C_VEL
LIN {X 0,Y 545.022,Z 49.595,A -85,B 0,C 180,E1 -3574.815,E2 -3574.815} C_VEL
LIN {X 0,Y 545.028,Z 49.593,A -85,B 0,C 180,E1 -3577.242,E2 -3577.242} C_VEL
LIN {X 0,Y 545.107,Z 49.581,A -85,B 0,C 180,E1 -3580.252,E2 -3580.252} C_VEL
LIN {X 0,Y 545.064,Z 49.59,A -85,B 0,C 180,E1 -3582.749,E2 -3582.749} C_VEL
LIN {X 0,Y 545.066,Z 49.584,A -85,B 0,C 180,E1 -3585.819,E2 -3585.819} C_VEL
LIN {X 0,Y 545.113,Z 49.583,A -85,B 0,C 180,E1 -3588.849,E2 -3588.849} C_VEL
LIN {X 0,Y 545.087,Z 49.583,A -85,B 0,C 180,E1 -3591.846,E2 -3591.846} C_VEL
LIN {X 0,Y 545.169,Z 49.574,A -85,B 0,C 180,E1 -3594.822,E2 -3594.822} C_VEL
LIN {X 0,Y 545.187,Z 49.572,A -85,B 0,C 180,E1 -3597.783,E2 -3597.783} C_VEL
LIN {X 0,Y 545.21,Z 49.567,A -85,B 0,C 180,E1 -3600.738,E2 -3600.738} C_VEL
LIN {X 0,Y 545.155,Z 49.573,A -85,B 0,C 180,E1 -3602.956,E2 -3602.956} C_VEL
LIN {X 0,Y 545.133,Z 49.581,A -85,B 0,C 180,E1 -3605.92,E2 -3605.92} C_VEL
LIN {X 0,Y 545.099,Z 49.58,A -85,B 0,C 180,E1 -3608.9,E2 -3608.9} C_VEL
LIN {X 0,Y 545.104,Z 49.585,A -85,B 0,C 180,E1 -3611.905,E2 -3611.905} C_VEL
LIN {X 0,Y 545.083,Z 49.583,A -85,B 0,C 180,E1 -3614.944,E2 -3614.944} C_VEL
LIN {X 0,Y 545.058,Z 49.587,A -85,B 0,C 180,E1 -3618.026,E2 -3618.026} C_VEL
LIN {X 0,Y 545.093,Z 49.581,A -85,B 0,C 180,E1 -3620.372,E2 -3620.372} C_VEL
LIN {X 0,Y 545.076,Z 49.589,A -85,B 0,C 180,E1 -3623.56,E2 -3623.56} C_VEL
LIN {X 0,Y 545.065,Z 49.584,A -85,B 0,C 180,E1 -3626.001,E2 -3626.001} C_VEL
LIN {X 0,Y 545.073,Z 49.587,A -85,B 0,C 180,E1 -3628.744,E2 -3628.744} C_VEL
LIN {X 0,Y 545.061,Z 49.586,A -85,B 0,C 180,E1 -3631.679,E2 -3631.679} C_VEL
LIN {X 0,Y 545.075,Z 49.587,A -85,B 0,C 180,E1 -3634.564,E2 -3634.564} C_VEL
LIN {X 0,Y 545.038,Z 49.589,A -85,B 0,C 180,E1 -3637.304,E2 -3637.304} C_VEL
LIN {X 0,Y 545.067,Z 49.586,A -85,B 0,C 180,E1 -3640.143,E2 -3640.143} C_VEL
LIN {X 0,Y 545.081,Z 49.585,A -85,B 0,C 180,E1 -3643.106,E2 -3643.106} C_VEL
LIN {X 0,Y 545.052,Z 49.59,A -85,B 0,C 180,E1 -3646.226,E2 -3646.226} C_VEL
LIN {X 0,Y 545.084,Z 49.585,A -85,B 0,C 180,E1 -3648.885,E2 -3648.885} C_VEL
LIN {X 0,Y 545.085,Z 49.585,A -85,B 0,C 180,E1 -3650.818,E2 -3650.818} C_VEL
LIN {X 0,Y 545.045,Z 49.589,A -85,B 0,C 180,E1 -3653.62,E2 -3653.62} C_VEL
LIN {X 0,Y 545.069,Z 49.593,A -85,B 0,C 180,E1 -3656.328,E2 -3656.328} C_VEL
LIN {X 0,Y 545.069,Z 49.587,A -85,B 0,C 180,E1 -3658.952,E2 -3658.952} C_VEL
LIN {X 0,Y 545.088,Z 49.586,A -85,B 0,C 180,E1 -3661.507,E2 -3661.507} C_VEL
LIN {X 0,Y 545.098,Z 49.584,A -85,B 0,C 180,E1 -3664.491,E2 -3664.491} C_VEL
LIN {X 0,Y 545.104,Z 49.625,A -85,B 0,C 180,E1 -3665.582,E2 -3665.582} C_VEL
LIN {X 0,Y 546.171,Z 56.764,A -85,B 0,C 180,E1 -3666.691,E2 -3666.691} C_VEL
LIN {X 0,Y 545.946,Z 70.296,A -85,B 0,C 180,E1 -3668.674,E2 -3668.674} C_VEL
LIN {X 0,Y 545.699,Z 87.87,A -85,B 0,C 180,E1 -3671.217,E2 -3671.217} C_VEL
LIN {X 0,Y 545.392,Z 108.117,A -85,B 0,C 180,E1 -3674.107,E2 -3674.107} C_VEL
LIN {X 0,Y 545.314,Z 117.631,A -85,B 0,C 180,E1 -3675.439,E2 -3675.439} C_VEL
LIN {X 0,Y 546.488,Z 127.11,A -85,B 0,C 180,E1 -3675.596,E2 -3675.596} C_VEL
LIN {X 0,Y 546.191,Z 225.995,A -85,B 0,C 180,E1 -3676.915,E2 -3676.915} C_VEL
LIN {X 0,Y 546.023,Z 239.31,A -85,B 0,C 180,E1 -3677.242,E2 -3677.242} C_VEL
LIN {X 0,Y 545.871,Z 252.636,A -85,B 0,C 180,E1 -3677.735,E2 -3677.735} C_VEL
LIN {X 0,Y 545.625,Z 264.237,A -85,B 0,C 180,E1 -3678.32,E2 -3678.32} C_VEL
LIN {X 0,Y 545.438,Z 275.451,A -85,B 0,C 180,E1 -3679.044,E2 -3679.044} C_VEL
LIN {X 0,Y 545.199,Z 285.925,A -85,B 0,C 180,E1 -3679.884,E2 -3679.884} C_VEL
LIN {X 0,Y 545.065,Z 294.494,A -85,B 0,C 180,E1 -3680.725,E2 -3680.725} C_VEL
LIN {X 0,Y 544.934,Z 302.402,A -85,B 0,C 180,E1 -3681.657,E2 -3681.657} C_VEL
LIN {X 0,Y 544.824,Z 310.127,A -85,B 0,C 180,E1 -3682.774,E2 -3682.774} C_VEL
LIN {X 0,Y 544.762,Z 317.25,A -85,B 0,C 180,E1 -3684.076,E2 -3684.076} C_VEL
LIN {X 0,Y 544.627,Z 321.985,A -85,B 0,C 180,E1 -3685.188,E2 -3685.188} C_VEL
LIN {X 0,Y 544.669,Z 325.609,A -85,B 0,C 180,E1 -3686.301,E2 -3686.301} C_VEL
LIN {X 0,Y 544.65,Z 327.476,A -85,B 0,C 180,E1 -3687.041,E2 -3687.041} C_VEL
LIN {X 0,Y 544.55,Z 329.872,A -85,B 0,C 180,E1 -3688.521,E2 -3688.521} C_VEL
LIN {X 0,Y 544.547,Z 330.483,A -85,B 0,C 180,E1 -3689.26,E2 -3689.26} C_VEL
LIN {X 0,Y 544.547,Z 330.701,A -85,B 0,C 180,E1 -3690,E2 -3690} C_VEL
LIN {X 0,Y 544.547,Z 330.484,A -85,B 0,C 180,E1 -3690.739,E2 -3690.739} C_VEL
LIN {X 0,Y 544.571,Z 328.879,A -85,B 0,C 180,E1 -3692.219,E2 -3692.219} C_VEL
LIN {X 0,Y 544.65,Z 327.483,A -85,B 0,C 180,E1 -3692.958,E2 -3692.958} C_VEL
LIN {X 0,Y 544.683,Z 324.54,A -85,B 0,C 180,E1 -3694.069,E2 -3694.069} C_VEL
LIN {X 0,Y 544.653,Z 320.553,A -85,B 0,C 180,E1 -3695.182,E2 -3695.182} C_VEL
LIN {X 0,Y 544.703,Z 315.278,A -85,B 0,C 180,E1 -3696.325,E2 -3696.325} C_VEL
LIN {X 0,Y 544.829,Z 308.972,A -85,B 0,C 180,E1 -3697.411,E2 -3697.411} C_VEL
LIN {X 0,Y 544.967,Z 300.921,A -85,B 0,C 180,E1 -3698.529,E2 -3698.529} C_VEL
LIN {X 0,Y 545.085,Z 292.717,A -85,B 0,C 180,E1 -3699.462,E2 -3699.462} C_VEL
LIN {X 0,Y 545.335,Z 282.721,A -85,B 0,C 180,E1 -3700.394,E2 -3700.394} C_VEL
LIN {X 0,Y 545.505,Z 271.861,A -85,B 0,C 180,E1 -3701.208,E2 -3701.208} C_VEL
LIN {X 0,Y 545.704,Z 260.378,A -85,B 0,C 180,E1 -3701.891,E2 -3701.891} C_VEL
LIN {X 0,Y 545.92,Z 248.133,A -85,B 0,C 180,E1 -3702.453,E2 -3702.453} C_VEL
LIN {X 0,Y 546.075,Z 235.289,A -85,B 0,C 180,E1 -3702.874,E2 -3702.874} C_VEL
LIN {X 0,Y 546.256,Z 221.681,A -85,B 0,C 180,E1 -3703.153,E2 -3703.153} C_VEL
LIN {X 0,Y 546.321,Z 124.546,A -85,B 0,C 180,E1 -3704.442,E2 -3704.442} C_VEL
LIN {X 0,Y 545.29,Z 117.414,A -85,B 0,C 180,E1 -3704.579,E2 -3704.579} C_VEL
LIN {X 0,Y 545.569,Z 97.096,A -85,B 0,C 180,E1 -3707.467,E2 -3707.467} C_VEL
LIN {X 0,Y 545.91,Z 77.117,A -85,B 0,C 180,E1 -3710.34,E2 -3710.34} C_VEL
LIN {X 0,Y 546.204,Z 58.203,A -85,B 0,C 180,E1 -3713.106,E2 -3713.106} C_VEL
LIN {X 0,Y 545.93,Z 53.816,A -85,B 0,C 180,E1 -3713.769,E2 -3713.769} C_VEL
LIN {X 0,Y 545.108,Z 49.587,A -85,B 0,C 180,E1 -3714.468,E2 -3714.468} C_VEL
LIN {X 0,Y 545.091,Z 49.587,A -85,B 0,C 180,E1 -3717.656,E2 -3717.656} C_VEL
LIN {X 0,Y 545.079,Z 49.588,A -85,B 0,C 180,E1 -3720.246,E2 -3720.246} C_VEL
LIN {X 0,Y 545.08,Z 49.582,A -85,B 0,C 180,E1 -3723.062,E2 -3723.062} C_VEL
LIN {X 0,Y 545.035,Z 49.595,A -85,B 0,C 180,E1 -3725.673,E2 -3725.673} C_VEL
LIN {X 0,Y 545.055,Z 49.588,A -85,B 0,C 180,E1 -3728.237,E2 -3728.237} C_VEL
LIN {X 0,Y 545.083,Z 49.582,A -85,B 0,C 180,E1 -3730.473,E2 -3730.473} C_VEL
LIN {X 0,Y 545.079,Z 49.585,A -85,B 0,C 180,E1 -3733.106,E2 -3733.106} C_VEL
LIN {X 0,Y 545.049,Z 49.587,A -85,B 0,C 180,E1 -3736.226,E2 -3736.226} C_VEL
LIN {X 0,Y 545.081,Z 49.584,A -85,B 0,C 180,E1 -3738.885,E2 -3738.885} C_VEL
LIN {X 0,Y 545.078,Z 49.585,A -85,B 0,C 180,E1 -3740.818,E2 -3740.818} C_VEL
LIN {X 0,Y 545.043,Z 49.591,A -85,B 0,C 180,E1 -3743.62,E2 -3743.62} C_VEL
LIN {X 0,Y 545.067,Z 49.584,A -85,B 0,C 180,E1 -3746.328,E2 -3746.328} C_VEL
LIN {X 0,Y 545.066,Z 49.592,A -85,B 0,C 180,E1 -3748.952,E2 -3748.952} C_VEL
LIN {X 0,Y 545.101,Z 49.582,A -85,B 0,C 180,E1 -3751.508,E2 -3751.508} C_VEL
LIN {X 0,Y 545.096,Z 49.584,A -85,B 0,C 180,E1 -3754.491,E2 -3754.491} C_VEL
LIN {X 0,Y 545.035,Z 49.591,A -85,B 0,C 180,E1 -3757.242,E2 -3757.242} C_VEL
LIN {X 0,Y 545.116,Z 49.583,A -85,B 0,C 180,E1 -3760.415,E2 -3760.415} C_VEL
LIN {X 0,Y 545.062,Z 49.585,A -85,B 0,C 180,E1 -3763.521,E2 -3763.521} C_VEL
LIN {X 0,Y 545.09,Z 49.582,A -85,B 0,C 180,E1 -3765.82,E2 -3765.82} C_VEL
LIN {X 0,Y 545.117,Z 49.581,A -85,B 0,C 180,E1 -3768.849,E2 -3768.849} C_VEL
LIN {X 0,Y 545.125,Z 49.579,A -85,B 0,C 180,E1 -3771.847,E2 -3771.847} C_VEL
LIN {X 0,Y 545.198,Z 49.569,A -85,B 0,C 180,E1 -3774.823,E2 -3774.823} C_VEL
LIN {X 0,Y 545.196,Z 49.572,A -85,B 0,C 180,E1 -3777.784,E2 -3777.784} C_VEL
LIN {X 0,Y 545.206,Z 49.568,A -85,B 0,C 180,E1 -3780.739,E2 -3780.739} C_VEL
LIN {X 0,Y 545.165,Z 49.572,A -85,B 0,C 180,E1 -3782.956,E2 -3782.956} C_VEL
LIN {X 0,Y 545.163,Z 49.581,A -85,B 0,C 180,E1 -3785.92,E2 -3785.92} C_VEL
LIN {X 0,Y 545.102,Z 49.58,A -85,B 0,C 180,E1 -3788.901,E2 -3788.901} C_VEL
LIN {X 0,Y 545.105,Z 49.586,A -85,B 0,C 180,E1 -3791.905,E2 -3791.905} C_VEL
LIN {X 0,Y 545.082,Z 49.583,A -85,B 0,C 180,E1 -3794.944,E2 -3794.944} C_VEL
LIN {X 0,Y 545.061,Z 49.587,A -85,B 0,C 180,E1 -3798.027,E2 -3798.027} C_VEL
LIN {X 0,Y 545.091,Z 49.581,A -85,B 0,C 180,E1 -3800.373,E2 -3800.373} C_VEL
LIN {X 0,Y 545.072,Z 49.589,A -85,B 0,C 180,E1 -3803.56,E2 -3803.56} C_VEL
LIN {X 0,Y 545.068,Z 49.584,A -85,B 0,C 180,E1 -3806.001,E2 -3806.001} C_VEL
LIN {X 0,Y 545.075,Z 49.586,A -85,B 0,C 180,E1 -3808.745,E2 -3808.745} C_VEL
LIN {X 0,Y 545.059,Z 49.587,A -85,B 0,C 180,E1 -3811.679,E2 -3811.679} C_VEL
LIN {X 0,Y 545.059,Z 49.588,A -85,B 0,C 180,E1 -3814.565,E2 -3814.565} C_VEL
LIN {X 0,Y 545.064,Z 49.593,A -85,B 0,C 180,E1 -3816.981,E2 -3816.981} C_VEL
LIN {X 0,Y 544.355,Z 49.676,A -85,B 0,C 180,E1 -3817.598,E2 -3817.598} C_VEL
LIN {X 0,Y 541.489,Z 50.035,A -85,B 0,C 180,E1 -3818.598,E2 -3818.598} C_VEL
LIN {X 0,Y 539.095,Z 50.33,A -85,B 0,C 180,E1 -3819.404,E2 -3819.404} C_VEL
LIN {X 0,Y 538.072,Z 50.456,A -85,B 0,C 180,E1 -3820.026,E2 -3820.026} C_VEL
LIN {X 0,Y 537.99,Z 50.467,A -85,B 0,C 180,E1 -3820.237,E2 -3820.237} C_VEL
LIN {X 0,Y 537.981,Z 50.472,A -85,B 0,C 180,E1 -3822.983,E2 -3822.983} C_VEL
LIN {X 0,Y 538.02,Z 50.463,A -85,B 0,C 180,E1 -3825.927,E2 -3825.927} C_VEL
LIN {X 0,Y 538.024,Z 50.462,A -85,B 0,C 180,E1 -3829.256,E2 -3829.256} C_VEL
LIN {X 0,Y 537.987,Z 50.47,A -85,B 0,C 180,E1 -3832.122,E2 -3832.122} C_VEL
LIN {X 0,Y 537.991,Z 50.467,A -85,B 0,C 180,E1 -3834.915,E2 -3834.915} C_VEL
LIN {X 0,Y 538.02,Z 50.463,A -85,B 0,C 180,E1 -3837.618,E2 -3837.618} C_VEL
LIN {X 0,Y 538.016,Z 50.471,A -85,B 0,C 180,E1 -3840.239,E2 -3840.239} C_VEL
LIN {X 0,Y 538.006,Z 50.464,A -85,B 0,C 180,E1 -3842.793,E2 -3842.793} C_VEL
LIN {X 0,Y 537.989,Z 50.466,A -85,B 0,C 180,E1 -3845.29,E2 -3845.29} C_VEL
LIN {X 0,Y 538.02,Z 50.47,A -85,B 0,C 180,E1 -3848.042,E2 -3848.042} C_VEL
LIN {X 0,Y 538.085,Z 50.459,A -85,B 0,C 180,E1 -3850.148,E2 -3850.148} C_VEL
LIN {X 0,Y 537.992,Z 50.468,A -85,B 0,C 180,E1 -3853.298,E2 -3853.298} C_VEL
LIN {X 0,Y 538.057,Z 50.467,A -85,B 0,C 180,E1 -3855.631,E2 -3855.631} C_VEL
LIN {X 0,Y 538.065,Z 50.482,A -85,B 0,C 180,E1 -3858.082,E2 -3858.082} C_VEL
LIN {X 0,Y 538.494,Z 55.509,A -85,B 0,C 180,E1 -3859.092,E2 -3859.092} C_VEL
LIN {X 0,Y 538.339,Z 67.12,A -85,B 0,C 180,E1 -3861.366,E2 -3861.366} C_VEL
LIN {X 0,Y 538.265,Z 71.881,A -85,B 0,C 180,E1 -3862.29,E2 -3862.29} C_VEL
LIN {X 0,Y 539.692,Z 80.363,A -85,B 0,C 180,E1 -3862.466,E2 -3862.466} C_VEL
LIN {X 0,Y 539.273,Z 178.938,A -85,B 0,C 180,E1 -3863.805,E2 -3863.805} C_VEL
LIN {X 0,Y 539.132,Z 192.551,A -85,B 0,C 180,E1 -3864.155,E2 -3864.155} C_VEL
LIN {X 0,Y 539.032,Z 204.774,A -85,B 0,C 180,E1 -3864.623,E2 -3864.623} C_VEL
LIN {X 0,Y 538.863,Z 216.513,A -85,B 0,C 180,E1 -3865.231,E2 -3865.231} C_VEL
LIN {X 0,Y 538.597,Z 227.792,A -85,B 0,C 180,E1 -3865.978,E2 -3865.978} C_VEL
LIN {X 0,Y 538.36,Z 237.972,A -85,B 0,C 180,E1 -3866.82,E2 -3866.82} C_VEL
LIN {X 0,Y 538.166,Z 247.15,A -85,B 0,C 180,E1 -3867.755,E2 -3867.755} C_VEL
LIN {X 0,Y 537.913,Z 256.051,A -85,B 0,C 180,E1 -3868.877,E2 -3868.877} C_VEL
LIN {X 0,Y 537.828,Z 263.228,A -85,B 0,C 180,E1 -3870,E2 -3870} C_VEL
LIN {X 0,Y 537.672,Z 269.006,A -85,B 0,C 180,E1 -3871.124,E2 -3871.124} C_VEL
LIN {X 0,Y 537.572,Z 273.568,A -85,B 0,C 180,E1 -3872.248,E2 -3872.248} C_VEL
LIN {X 0,Y 537.596,Z 275.989,A -85,B 0,C 180,E1 -3872.998,E2 -3872.998} C_VEL
LIN {X 0,Y 537.567,Z 277.966,A -85,B 0,C 180,E1 -3873.748,E2 -3873.748} C_VEL
LIN {X 0,Y 537.517,Z 279.539,A -85,B 0,C 180,E1 -3874.5,E2 -3874.5} C_VEL
LIN {X 0,Y 537.526,Z 280.702,A -85,B 0,C 180,E1 -3875.251,E2 -3875.251} C_VEL
LIN {X 0,Y 537.59,Z 281.716,A -85,B 0,C 180,E1 -3876.502,E2 -3876.502} C_VEL
LIN {X 0,Y 537.52,Z 281.736,A -85,B 0,C 180,E1 -3877.513,E2 -3877.513} C_VEL
LIN {X 0,Y 537.527,Z 281.305,A -85,B 0,C 180,E1 -3878.269,E2 -3878.269} C_VEL
LIN {X 0,Y 537.524,Z 279.166,A -85,B 0,C 180,E1 -3879.786,E2 -3879.786} C_VEL
LIN {X 0,Y 537.597,Z 276.459,A -85,B 0,C 180,E1 -3880.927,E2 -3880.927} C_VEL
LIN {X 0,Y 537.649,Z 272.709,A -85,B 0,C 180,E1 -3882.073,E2 -3882.073} C_VEL
LIN {X 0,Y 537.699,Z 267.797,A -85,B 0,C 180,E1 -3883.223,E2 -3883.223} C_VEL
LIN {X 0,Y 537.827,Z 261.567,A -85,B 0,C 180,E1 -3884.376,E2 -3884.376} C_VEL
LIN {X 0,Y 537.987,Z 253.736,A -85,B 0,C 180,E1 -3885.534,E2 -3885.534} C_VEL
LIN {X 0,Y 538.147,Z 245.657,A -85,B 0,C 180,E1 -3886.502,E2 -3886.502} C_VEL
LIN {X 0,Y 538.391,Z 235.737,A -85,B 0,C 180,E1 -3887.472,E2 -3887.472} C_VEL
LIN {X 0,Y 538.597,Z 225.947,A -85,B 0,C 180,E1 -3888.251,E2 -3888.251} C_VEL
LIN {X 0,Y 538.811,Z 215.338,A -85,B 0,C 180,E1 -3888.933,E2 -3888.933} C_VEL
LIN {X 0,Y 539.034,Z 203.616,A -85,B 0,C 180,E1 -3889.518,E2 -3889.518} C_VEL
LIN {X 0,Y 539.212,Z 190.28,A -85,B 0,C 180,E1 -3890.006,E2 -3890.006} C_VEL
LIN {X 0,Y 539.352,Z 177.148,A -85,B 0,C 180,E1 -3890.318,E2 -3890.318} C_VEL
LIN {X 0,Y 539.639,Z 79.094,A -85,B 0,C 180,E1 -3891.643,E2 -3891.643} C_VEL
LIN {X 0,Y 538.286,Z 72.003,A -85,B 0,C 180,E1 -3891.785,E2 -3891.785} C_VEL
LIN {X 0,Y 538.5,Z 56.1,A -85,B 0,C 180,E1 -3894.891,E2 -3894.891} C_VEL
LIN {X 0,Y 538.049,Z 50.467,A -85,B 0,C 180,E1 -3896.049,E2 -3896.049} C_VEL
LIN {X 0,Y 537.997,Z 50.469,A -85,B 0,C 180,E1 -3898.926,E2 -3898.926} C_VEL
LIN {X 0,Y 538,Z 50.47,A -85,B 0,C 180,E1 -3901.884,E2 -3901.884} C_VEL
LIN {X 0,Y 537.995,Z 50.469,A -85,B 0,C 180,E1 -3904.614,E2 -3904.614} C_VEL
LIN {X 0,Y 537.973,Z 50.474,A -85,B 0,C 180,E1 -3907.88,E2 -3907.88} C_VEL
LIN {X 0,Y 537.955,Z 50.471,A -85,B 0,C 180,E1 -3910.785,E2 -3910.785} C_VEL
LIN {X 0,Y 537.981,Z 50.473,A -85,B 0,C 180,E1 -3913.819,E2 -3913.819} C_VEL
LIN {X 0,Y 537.982,Z 50.47,A -85,B 0,C 180,E1 -3916.181,E2 -3916.181} C_VEL
LIN {X 0,Y 537.954,Z 50.473,A -85,B 0,C 180,E1 -3919.265,E2 -3919.265} C_VEL
LIN {X 0,Y 537.95,Z 50.473,A -85,B 0,C 180,E1 -3922.118,E2 -3922.118} C_VEL
LIN {X 0,Y 537.994,Z 50.473,A -85,B 0,C 180,E1 -3925.386,E2 -3925.386} C_VEL
LIN {X 0,Y 537.998,Z 50.464,A -85,B 0,C 180,E1 -3928.116,E2 -3928.116} C_VEL
LIN {X 0,Y 537.987,Z 50.474,A -85,B 0,C 180,E1 -3931.095,E2 -3931.095} C_VEL
LIN {X 0,Y 537.972,Z 50.47,A -85,B 0,C 180,E1 -3933.629,E2 -3933.629} C_VEL
LIN {X 0,Y 538.009,Z 50.463,A -85,B 0,C 180,E1 -3936.122,E2 -3936.122} C_VEL
LIN {X 0,Y 538.036,Z 50.463,A -85,B 0,C 180,E1 -3939.348,E2 -3939.348} C_VEL
LIN {X 0,Y 538.032,Z 50.464,A -85,B 0,C 180,E1 -3942.516,E2 -3942.516} C_VEL
LIN {X 0,Y 538.04,Z 50.46,A -85,B 0,C 180,E1 -3945.63,E2 -3945.63} C_VEL
LIN {X 0,Y 538.075,Z 50.462,A -85,B 0,C 180,E1 -3948.701,E2 -3948.701} C_VEL
LIN {X 0,Y 538.053,Z 50.459,A -85,B 0,C 180,E1 -3951.739,E2 -3951.739} C_VEL
LIN {X 0,Y 538.127,Z 50.451,A -85,B 0,C 180,E1 -3954.754,E2 -3954.754} C_VEL
LIN {X 0,Y 538.16,Z 50.447,A -85,B 0,C 180,E1 -3957.755,E2 -3957.755} C_VEL
LIN {X 0,Y 538.18,Z 50.442,A -85,B 0,C 180,E1 -3960.748,E2 -3960.748} C_VEL
LIN {X 0,Y 538.121,Z 50.45,A -85,B 0,C 180,E1 -3962.994,E2 -3962.994} C_VEL
LIN {X 0,Y 538.09,Z 50.458,A -85,B 0,C 180,E1 -3965.998,E2 -3965.998} C_VEL
LIN {X 0,Y 538.052,Z 50.458,A -85,B 0,C 180,E1 -3969.018,E2 -3969.018} C_VEL
LIN {X 0,Y 538.064,Z 50.459,A -85,B 0,C 180,E1 -3972.063,E2 -3972.063} C_VEL
LIN {X 0,Y 538.043,Z 50.461,A -85,B 0,C 180,E1 -3975.144,E2 -3975.144} C_VEL
LIN {X 0,Y 538.012,Z 50.463,A -85,B 0,C 180,E1 -3978.271,E2 -3978.271} C_VEL
LIN {X 0,Y 538.039,Z 50.46,A -85,B 0,C 180,E1 -3980.651,E2 -3980.651} C_VEL
LIN {X 0,Y 538.009,Z 50.465,A -85,B 0,C 180,E1 -3983.877,E2 -3983.877} C_VEL
LIN {X 0,Y 538.032,Z 50.46,A -85,B 0,C 180,E1 -3986.367,E2 -3986.367} C_VEL
LIN {X 0,Y 538.033,Z 50.466,A -85,B 0,C 180,E1 -3988.933,E2 -3988.933} C_VEL
LIN {X 0,Y 538.013,Z 50.463,A -85,B 0,C 180,E1 -3991.887,E2 -3991.887} C_VEL
LIN {X 0,Y 538.024,Z 50.466,A -85,B 0,C 180,E1 -3994.619,E2 -3994.619} C_VEL
LIN {X 0,Y 538.006,Z 50.466,A -85,B 0,C 180,E1 -3997.17,E2 -3997.17} C_VEL
LIN {X 0,Y 538.024,Z 50.462,A -85,B 0,C 180,E1 -3999.797,E2 -3999.797} C_VEL
LIN {X 0,Y 538.022,Z 50.469,A -85,B 0,C 180,E1 -4002.786,E2 -4002.786} C_VEL
LIN {X 0,Y 538.021,Z 50.463,A -85,B 0,C 180,E1 -4005.927,E2 -4005.927} C_VEL
LIN {X 0,Y 538.033,Z 50.466,A -85,B 0,C 180,E1 -4008.227,E2 -4008.227} C_VEL
LIN {X 0,Y 538.017,Z 50.463,A -85,B 0,C 180,E1 -4011.17,E2 -4011.17} C_VEL
LIN {X 0,Y 537.997,Z 50.472,A -85,B 0,C 180,E1 -4014.089,E2 -4014.089} C_VEL
LIN {X 0,Y 538.034,Z 50.465,A -85,B 0,C 180,E1 -4016.727,E2 -4016.727} C_VEL
LIN {X 0,Y 538.03,Z 50.466,A -85,B 0,C 180,E1 -4019.556,E2 -4019.556} C_VEL
LIN {X 0,Y 538.06,Z 50.46,A -85,B 0,C 180,E1 -4022.648,E2 -4022.648} C_VEL
LIN {X 0,Y 538.105,Z 50.627,A -85,B 0,C 180,E1 -4025.436,E2 -4025.436} C_VEL
LIN {X 0,Y 539.228,Z 57.843,A -85,B 0,C 180,E1 -4026.576,E2 -4026.576} C_VEL
LIN {X 0,Y 538.993,Z 71.344,A -85,B 0,C 180,E1 -4028.586,E2 -4028.586} C_VEL
LIN {X 0,Y 538.689,Z 88.91,A -85,B 0,C 180,E1 -4031.161,E2 -4031.161} C_VEL
LIN {X 0,Y 538.377,Z 107.786,A -85,B 0,C 180,E1 -4033.895,E2 -4033.895} C_VEL
LIN {X 0,Y 538.241,Z 117.151,A -85,B 0,C 180,E1 -4035.24,E2 -4035.24} C_VEL
LIN {X 0,Y 539.605,Z 127.489,A -85,B 0,C 180,E1 -4035.418,E2 -4035.418} C_VEL
LIN {X 0,Y 539.287,Z 225.655,A -85,B 0,C 180,E1 -4036.745,E2 -4036.745} C_VEL
LIN {X 0,Y 539.108,Z 238.975,A -85,B 0,C 180,E1 -4037.076,E2 -4037.076} C_VEL
LIN {X 0,Y 538.899,Z 251.175,A -85,B 0,C 180,E1 -4037.526,E2 -4037.526} C_VEL
LIN {X 0,Y 538.675,Z 263.201,A -85,B 0,C 180,E1 -4038.125,E2 -4038.125} C_VEL
LIN {X 0,Y 538.433,Z 275.12,A -85,B 0,C 180,E1 -4038.899,E2 -4038.899} C_VEL
LIN {X 0,Y 538.19,Z 285.596,A -85,B 0,C 180,E1 -4039.751,E2 -4039.751} C_VEL
LIN {X 0,Y 538.023,Z 294.165,A -85,B 0,C 180,E1 -4040.602,E2 -4040.602} C_VEL
LIN {X 0,Y 537.884,Z 302.075,A -85,B 0,C 180,E1 -4041.547,E2 -4041.547} C_VEL
LIN {X 0,Y 537.752,Z 309.801,A -85,B 0,C 180,E1 -4042.679,E2 -4042.679} C_VEL
LIN {X 0,Y 537.649,Z 316.924,A -85,B 0,C 180,E1 -4043.997,E2 -4043.997} C_VEL
LIN {X 0,Y 537.539,Z 321.661,A -85,B 0,C 180,E1 -4045.125,E2 -4045.125} C_VEL
LIN {X 0,Y 537.591,Z 325.286,A -85,B 0,C 180,E1 -4046.252,E2 -4046.252} C_VEL
LIN {X 0,Y 537.58,Z 327.155,A -85,B 0,C 180,E1 -4047.002,E2 -4047.002} C_VEL
LIN {X 0,Y 537.456,Z 329.551,A -85,B 0,C 180,E1 -4048.501,E2 -4048.501} C_VEL
LIN {X 0,Y 537.454,Z 330.162,A -85,B 0,C 180,E1 -4049.251,E2 -4049.251} C_VEL
LIN {X 0,Y 537.455,Z 330.38,A -85,B 0,C 180,E1 -4050,E2 -4050} C_VEL
LIN {X 0,Y 537.454,Z 330.164,A -85,B 0,C 180,E1 -4050.749,E2 -4050.749} C_VEL
LIN {X 0,Y 537.49,Z 328.56,A -85,B 0,C 180,E1 -4052.248,E2 -4052.248} C_VEL
LIN {X 0,Y 537.58,Z 327.164,A -85,B 0,C 180,E1 -4052.997,E2 -4052.997} C_VEL
LIN {X 0,Y 537.602,Z 324.221,A -85,B 0,C 180,E1 -4054.123,E2 -4054.123} C_VEL
LIN {X 0,Y 537.587,Z 320.234,A -85,B 0,C 180,E1 -4055.25,E2 -4055.25} C_VEL
LIN {X 0,Y 537.641,Z 314.188,A -85,B 0,C 180,E1 -4056.552,E2 -4056.552} C_VEL
LIN {X 0,Y 537.774,Z 307.41,A -85,B 0,C 180,E1 -4057.698,E2 -4057.698} C_VEL
LIN {X 0,Y 537.919,Z 299.103,A -85,B 0,C 180,E1 -4058.83,E2 -4058.83} C_VEL
LIN {X 0,Y 538.065,Z 290.59,A -85,B 0,C 180,E1 -4059.776,E2 -4059.776} C_VEL
LIN {X 0,Y 538.321,Z 280.076,A -85,B 0,C 180,E1 -4060.722,E2 -4060.722} C_VEL
LIN {X 0,Y 538.548,Z 268.975,A -85,B 0,C 180,E1 -4061.526,E2 -4061.526} C_VEL
LIN {X 0,Y 538.773,Z 258.281,A -85,B 0,C 180,E1 -4062.142,E2 -4062.142} C_VEL
LIN {X 0,Y 538.982,Z 246.592,A -85,B 0,C 180,E1 -4062.663,E2 -4062.663} C_VEL
LIN {X 0,Y 539.177,Z 233.129,A -85,B 0,C 180,E1 -4063.09,E2 -4063.09} C_VEL
LIN {X 0,Y 539.378,Z 219.826,A -85,B 0,C 180,E1 -4063.348,E2 -4063.348} C_VEL
LIN {X 0,Y 539.551,Z 126.01,A -85,B 0,C 180,E1 -4064.604,E2 -4064.604} C_VEL
LIN {X 0,Y 538.229,Z 117.062,A -85,B 0,C 180,E1 -4064.779,E2 -4064.779} C_VEL
LIN {X 0,Y 538.561,Z 98.401,A -85,B 0,C 180,E1 -4067.466,E2 -4067.466} C_VEL
LIN {X 0,Y 538.921,Z 76.821,A -85,B 0,C 180,E1 -4070.616,E2 -4070.616} C_VEL
LIN {X 0,Y 539.27,Z 59.257,A -85,B 0,C 180,E1 -4073.218,E2 -4073.218} C_VEL
LIN {X 0,Y 538.995,Z 55.176,A -85,B 0,C 180,E1 -4073.841,E2 -4073.841} C_VEL
LIN {X 0,Y 538.063,Z 50.464,A -85,B 0,C 180,E1 -4074.613,E2 -4074.613} C_VEL
LIN {X 0,Y 538.059,Z 50.46,A -85,B 0,C 180,E1 -4077.352,E2 -4077.352} C_VEL
LIN {X 0,Y 538.019,Z 50.469,A -85,B 0,C 180,E1 -4079.761,E2 -4079.761} C_VEL
LIN {X 0,Y 538.02,Z 50.464,A -85,B 0,C 180,E1 -4082.382,E2 -4082.382} C_VEL
LIN {X 0,Y 538,Z 50.465,A -85,B 0,C 180,E1 -4085.084,E2 -4085.084} C_VEL
LIN {X 0,Y 537.994,Z 50.472,A -85,B 0,C 180,E1 -4087.877,E2 -4087.877} C_VEL
LIN {X 0,Y 538.049,Z 50.458,A -85,B 0,C 180,E1 -4090.776,E2 -4090.776} C_VEL
LIN {X 0,Y 538.003,Z 50.469,A -85,B 0,C 180,E1 -4093.816,E2 -4093.816} C_VEL
LIN {X 0,Y 538.026,Z 50.464,A -85,B 0,C 180,E1 -4097.012,E2 -4097.012} C_VEL
LIN {X 0,Y 538.048,Z 50.466,A -85,B 0,C 180,E1 -4099.253,E2 -4099.253} C_VEL
LIN {X 0,Y 537.99,Z 50.466,A -85,B 0,C 180,E1 -4102.122,E2 -4102.122} C_VEL
LIN {X 0,Y 538.007,Z 50.468,A -85,B 0,C 180,E1 -4104.916,E2 -4104.916} C_VEL
LIN {X 0,Y 538.019,Z 50.464,A -85,B 0,C 180,E1 -4107.617,E2 -4107.617} C_VEL
LIN {X 0,Y 538.015,Z 50.463,A -85,B 0,C 180,E1 -4110.239,E2 -4110.239} C_VEL
LIN {X 0,Y 538.057,Z 50.464,A -85,B 0,C 180,E1 -4112.796,E2 -4112.796} C_VEL
LIN {X 0,Y 538.027,Z 50.464,A -85,B 0,C 180,E1 -4115.292,E2 -4115.292} C_VEL
LIN {X 0,Y 538.015,Z 50.463,A -85,B 0,C 180,E1 -4118.042,E2 -4118.042} C_VEL
LIN {X 0,Y 538.032,Z 50.466,A -85,B 0,C 180,E1 -4120.94,E2 -4120.94} C_VEL
LIN {X 0,Y 538.01,Z 50.464,A -85,B 0,C 180,E1 -4123.299,E2 -4123.299} C_VEL
LIN {X 0,Y 538.06,Z 50.457,A -85,B 0,C 180,E1 -4125.631,E2 -4125.631} C_VEL
LIN {X 0,Y 538.077,Z 50.46,A -85,B 0,C 180,E1 -4128.702,E2 -4128.702} C_VEL
LIN {X 0,Y 538.082,Z 50.455,A -85,B 0,C 180,E1 -4131.74,E2 -4131.74} C_VEL
LIN {X 0,Y 538.121,Z 50.454,A -85,B 0,C 180,E1 -4134.003,E2 -4134.003} C_VEL
LIN {X 0,Y 538.133,Z 50.448,A -85,B 0,C 180,E1 -4137.006,E2 -4137.006} C_VEL
LIN {X 0,Y 538.174,Z 50.45,A -85,B 0,C 180,E1 -4140,E2 -4140} C_VEL
LIN {X 0,Y 538.133,Z 50.448,A -85,B 0,C 180,E1 -4142.995,E2 -4142.995} C_VEL
LIN {X 0,Y 538.114,Z 50.458,A -85,B 0,C 180,E1 -4145.998,E2 -4145.998} C_VEL
LIN {X 0,Y 538.054,Z 50.458,A -85,B 0,C 180,E1 -4149.018,E2 -4149.018} C_VEL
LIN {X 0,Y 538.064,Z 50.46,A -85,B 0,C 180,E1 -4152.063,E2 -4152.063} C_VEL
LIN {X 0,Y 538.042,Z 50.462,A -85,B 0,C 180,E1 -4155.144,E2 -4155.144} C_VEL
LIN {X 0,Y 538.014,Z 50.463,A -85,B 0,C 180,E1 -4158.271,E2 -4158.271} C_VEL
LIN {X 0,Y 538.037,Z 50.46,A -85,B 0,C 180,E1 -4160.652,E2 -4160.652} C_VEL
LIN {X 0,Y 538.006,Z 50.465,A -85,B 0,C 180,E1 -4163.878,E2 -4163.878} C_VEL
LIN {X 0,Y 538.036,Z 50.46,A -85,B 0,C 180,E1 -4166.367,E2 -4166.367} C_VEL
LIN {X 0,Y 538.031,Z 50.466,A -85,B 0,C 180,E1 -4168.934,E2 -4168.934} C_VEL
LIN {X 0,Y 538.01,Z 50.463,A -85,B 0,C 180,E1 -4171.887,E2 -4171.887} C_VEL
LIN {X 0,Y 538.009,Z 50.467,A -85,B 0,C 180,E1 -4174.617,E2 -4174.617} C_VEL
LIN {X 0,Y 538.004,Z 50.469,A -85,B 0,C 180,E1 -4177.17,E2 -4177.17} C_VEL
LIN {X 0,Y 538.01,Z 50.463,A -85,B 0,C 180,E1 -4179.799,E2 -4179.799} C_VEL
LIN {X 0,Y 537.99,Z 50.467,A -85,B 0,C 180,E1 -4180.237,E2 -4180.237} C_VEL
LIN {X 0,Y 537.327,Z 50.557,A -85,B 0,C 180,E1 -4180.862,E2 -4180.862} C_VEL
LIN {X 0,Y 534.477,Z 50.91,A -85,B 0,C 180,E1 -4181.877,E2 -4181.877} C_VEL
LIN {X 0,Y 532.063,Z 51.212,A -85,B 0,C 180,E1 -4182.694,E2 -4182.694} C_VEL
LIN {X 0,Y 531.024,Z 51.335,A -85,B 0,C 180,E1 -4183.324,E2 -4183.324} C_VEL
LIN {X 0,Y 530.938,Z 51.344,A -85,B 0,C 180,E1 -4183.538,E2 -4183.538} C_VEL
LIN {X 0,Y 530.946,Z 51.35,A -85,B 0,C 180,E1 -4186.504,E2 -4186.504} C_VEL
LIN {X 0,Y 530.963,Z 51.344,A -85,B 0,C 180,E1 -4188.98,E2 -4188.98} C_VEL
LIN {X 0,Y 530.953,Z 51.342,A -85,B 0,C 180,E1 -4191.529,E2 -4191.529} C_VEL
LIN {X 0,Y 530.949,Z 51.352,A -85,B 0,C 180,E1 -4194.38,E2 -4194.38} C_VEL
LIN {X 0,Y 530.97,Z 51.34,A -85,B 0,C 180,E1 -4197.134,E2 -4197.134} C_VEL
LIN {X 0,Y 530.971,Z 51.343,A -85,B 0,C 180,E1 -4199.803,E2 -4199.803} C_VEL
LIN {X 0,Y 530.966,Z 51.344,A -85,B 0,C 180,E1 -4202.478,E2 -4202.478} C_VEL
LIN {X 0,Y 530.953,Z 51.342,A -85,B 0,C 180,E1 -4204.94,E2 -4204.94} C_VEL
LIN {X 0,Y 530.982,Z 51.347,A -85,B 0,C 180,E1 -4207.899,E2 -4207.899} C_VEL
LIN {X 0,Y 530.985,Z 51.338,A -85,B 0,C 180,E1 -4210.677,E2 -4210.677} C_VEL
LIN {X 0,Y 530.958,Z 51.342,A -85,B 0,C 180,E1 -4213.07,E2 -4213.07} C_VEL
LIN {X 0,Y 531.017,Z 51.342,A -85,B 0,C 180,E1 -4215.436,E2 -4215.436} C_VEL
LIN {X 0,Y 531.04,Z 51.456,A -85,B 0,C 180,E1 -4217.983,E2 -4217.983} C_VEL
LIN {X 0,Y 531.5,Z 56.201,A -85,B 0,C 180,E1 -4218.946,E2 -4218.946} C_VEL
LIN {X 0,Y 531.368,Z 67.86,A -85,B 0,C 180,E1 -4221.251,E2 -4221.251} C_VEL
LIN {X 0,Y 531.265,Z 72.269,A -85,B 0,C 180,E1 -4222.112,E2 -4222.112} C_VEL
LIN {X 0,Y 532.849,Z 81.806,A -85,B 0,C 180,E1 -4222.29,E2 -4222.29} C_VEL
LIN {X 0,Y 532.381,Z 179.189,A -85,B 0,C 180,E1 -4223.629,E2 -4223.629} C_VEL
LIN {X 0,Y 532.221,Z 192.827,A -85,B 0,C 180,E1 -4223.984,E2 -4223.984} C_VEL
LIN {X 0,Y 532.112,Z 205.061,A -85,B 0,C 180,E1 -4224.458,E2 -4224.458} C_VEL
LIN {X 0,Y 531.928,Z 216.808,A -85,B 0,C 180,E1 -4225.074,E2 -4225.074} C_VEL
LIN {X 0,Y 531.639,Z 228.091,A -85,B 0,C 180,E1 -4225.831,E2 -4225.831} C_VEL
LIN {X 0,Y 531.372,Z 238.277,A -85,B 0,C 180,E1 -4226.683,E2 -4226.683} C_VEL
LIN {X 0,Y 531.193,Z 246.616,A -85,B 0,C 180,E1 -4227.536,E2 -4227.536} C_VEL
LIN {X 0,Y 530.899,Z 255.694,A -85,B 0,C 180,E1 -4228.673,E2 -4228.673} C_VEL
LIN {X 0,Y 530.8,Z 262.989,A -85,B 0,C 180,E1 -4229.811,E2 -4229.811} C_VEL
LIN {X 0,Y 530.608,Z 269.748,A -85,B 0,C 180,E1 -4231.139,E2 -4231.139} C_VEL
LIN {X 0,Y 530.496,Z 274.215,A -85,B 0,C 180,E1 -4232.278,E2 -4232.278} C_VEL
LIN {X 0,Y 530.525,Z 276.567,A -85,B 0,C 180,E1 -4233.038,E2 -4233.038} C_VEL
LIN {X 0,Y 530.487,Z 278.504,A -85,B 0,C 180,E1 -4233.798,E2 -4233.798} C_VEL
LIN {X 0,Y 530.426,Z 280.037,A -85,B 0,C 180,E1 -4234.56,E2 -4234.56} C_VEL
LIN {X 0,Y 530.453,Z 281.122,A -85,B 0,C 180,E1 -4235.322,E2 -4235.322} C_VEL
LIN {X 0,Y 530.522,Z 282.038,A -85,B 0,C 180,E1 -4236.507,E2 -4236.507} C_VEL
LIN {X 0,Y 530.431,Z 282.037,A -85,B 0,C 180,E1 -4237.614,E2 -4237.614} C_VEL
LIN {X 0,Y 530.438,Z 281.53,A -85,B 0,C 180,E1 -4238.381,E2 -4238.381} C_VEL
LIN {X 0,Y 530.447,Z 279.307,A -85,B 0,C 180,E1 -4239.918,E2 -4239.918} C_VEL
LIN {X 0,Y 530.481,Z 277.581,A -85,B 0,C 180,E1 -4240.689,E2 -4240.689} C_VEL
LIN {X 0,Y 530.578,Z 274.103,A -85,B 0,C 180,E1 -4241.848,E2 -4241.848} C_VEL
LIN {X 0,Y 530.623,Z 269.494,A -85,B 0,C 180,E1 -4243.013,E2 -4243.013} C_VEL
LIN {X 0,Y 530.792,Z 262.46,A -85,B 0,C 180,E1 -4244.375,E2 -4244.375} C_VEL
LIN {X 0,Y 530.937,Z 254.796,A -85,B 0,C 180,E1 -4245.548,E2 -4245.548} C_VEL
LIN {X 0,Y 531.133,Z 246.892,A -85,B 0,C 180,E1 -4246.529,E2 -4246.529} C_VEL
LIN {X 0,Y 531.374,Z 237.158,A -85,B 0,C 180,E1 -4247.512,E2 -4247.512} C_VEL
LIN {X 0,Y 531.577,Z 227.599,A -85,B 0,C 180,E1 -4248.301,E2 -4248.301} C_VEL
LIN {X 0,Y 531.874,Z 215.673,A -85,B 0,C 180,E1 -4249.089,E2 -4249.089} C_VEL
LIN {X 0,Y 532.118,Z 203.957,A -85,B 0,C 180,E1 -4249.682,E2 -4249.682} C_VEL
LIN {X 0,Y 532.32,Z 190.792,A -85,B 0,C 180,E1 -4250.17,E2 -4250.17} C_VEL
LIN {X 0,Y 532.475,Z 177.687,A -85,B 0,C 180,E1 -4250.489,E2 -4250.489} C_VEL
LIN {X 0,Y 532.699,Z 79.554,A -85,B 0,C 180,E1 -4251.836,E2 -4251.836} C_VEL
LIN {X 0,Y 531.303,Z 72.291,A -85,B 0,C 180,E1 -4251.984,E2 -4251.984} C_VEL
LIN {X 0,Y 531.526,Z 56.816,A -85,B 0,C 180,E1 -4255.032,E2 -4255.032} C_VEL
LIN {X 0,Y 530.977,Z 51.348,A -85,B 0,C 180,E1 -4256.163,E2 -4256.163} C_VEL
LIN {X 0,Y 530.964,Z 51.343,A -85,B 0,C 180,E1 -4259.324,E2 -4259.324} C_VEL
LIN {X 0,Y 530.955,Z 51.351,A -85,B 0,C 180,E1 -4262.098,E2 -4262.098} C_VEL
LIN {X 0,Y 530.956,Z 51.344,A -85,B 0,C 180,E1 -4264.848,E2 -4264.848} C_VEL
LIN {X 0,Y 530.929,Z 51.348,A -85,B 0,C 180,E1 -4267.511,E2 -4267.511} C_VEL
LIN {X 0,Y 530.909,Z 51.351,A -85,B 0,C 180,E1 -4270.44,E2 -4270.44} C_VEL
LIN {X 0,Y 530.923,Z 51.351,A -85,B 0,C 180,E1 -4273.499,E2 -4273.499} C_VEL
LIN {X 0,Y 530.966,Z 51.344,A -85,B 0,C 180,E1 -4275.624,E2 -4275.624} C_VEL
LIN {X 0,Y 530.909,Z 51.347,A -85,B 0,C 180,E1 -4278.556,E2 -4278.556} C_VEL
LIN {X 0,Y 530.913,Z 51.355,A -85,B 0,C 180,E1 -4281.525,E2 -4281.525} C_VEL
LIN {X 0,Y 530.929,Z 51.344,A -85,B 0,C 180,E1 -4284.378,E2 -4284.378} C_VEL
LIN {X 0,Y 530.948,Z 51.349,A -85,B 0,C 180,E1 -4287.132,E2 -4287.132} C_VEL
LIN {X 0,Y 530.933,Z 51.347,A -85,B 0,C 180,E1 -4289.8,E2 -4289.8} C_VEL
LIN {X 0,Y 530.958,Z 51.341,A -85,B 0,C 180,E1 -4292.48,E2 -4292.48} C_VEL
LIN {X 0,Y 530.948,Z 51.343,A -85,B 0,C 180,E1 -4295.774,E2 -4295.774} C_VEL
LIN {X 0,Y 530.998,Z 51.344,A -85,B 0,C 180,E1 -4299.062,E2 -4299.062} C_VEL
LIN {X 0,Y 530.971,Z 51.339,A -85,B 0,C 180,E1 -4301.478,E2 -4301.478} C_VEL
LIN {X 0,Y 530.987,Z 51.345,A -85,B 0,C 180,E1 -4304.65,E2 -4304.65} C_VEL
LIN {X 0,Y 531.019,Z 51.331,A -85,B 0,C 180,E1 -4307.774,E2 -4307.774} C_VEL
LIN {X 0,Y 530.969,Z 51.343,A -85,B 0,C 180,E1 -4310.092,E2 -4310.092} C_VEL
LIN {X 0,Y 531.022,Z 51.332,A -85,B 0,C 180,E1 -4313.034,E2 -4313.034} C_VEL
LIN {X 0,Y 530.979,Z 51.338,A -85,B 0,C 180,E1 -4315.445,E2 -4315.445} C_VEL
LIN {X 0,Y 531.133,Z 51.322,A -85,B 0,C 180,E1 -4317.725,E2 -4317.725} C_VEL
LIN {X 0,Y 531.151,Z 51.318,A -85,B 0,C 180,E1 -4320.758,E2 -4320.758} C_VEL
LIN {X 0,Y 531.062,Z 51.329,A -85,B 0,C 180,E1 -4323.034,E2 -4323.034} C_VEL
LIN {X 0,Y 531.049,Z 51.335,A -85,B 0,C 180,E1 -4326.077,E2 -4326.077} C_VEL
LIN {X 0,Y 531.014,Z 51.335,A -85,B 0,C 180,E1 -4329.138,E2 -4329.138} C_VEL
LIN {X 0,Y 531.053,Z 51.335,A -85,B 0,C 180,E1 -4331.67,E2 -4331.67} C_VEL
LIN {X 0,Y 531.026,Z 51.334,A -85,B 0,C 180,E1 -4334.952,E2 -4334.952} C_VEL
LIN {X 0,Y 530.975,Z 51.345,A -85,B 0,C 180,E1 -4337.724,E2 -4337.724} C_VEL
LIN {X 0,Y 531.028,Z 51.334,A -85,B 0,C 180,E1 -4340.127,E2 -4340.127} C_VEL
LIN {X 0,Y 530.945,Z 51.341,A -85,B 0,C 180,E1 -4342.573,E2 -4342.573} C_VEL
LIN {X 0,Y 530.964,Z 51.347,A -85,B 0,C 180,E1 -4345.06,E2 -4345.06} C_VEL
LIN {X 0,Y 531.011,Z 51.338,A -85,B 0,C 180,E1 -4347.596,E2 -4347.596} C_VEL
LIN {X 0,Y 530.964,Z 51.344,A -85,B 0,C 180,E1 -4350.642,E2 -4350.642} C_VEL
LIN {X 0,Y 530.991,Z 51.338,A -85,B 0,C 180,E1 -4353.772,E2 -4353.772} C_VEL
LIN {X 0,Y 530.958,Z 51.341,A -85,B 0,C 180,E1 -4356.558,E2 -4356.558} C_VEL
LIN {X 0,Y 530.987,Z 51.34,A -85,B 0,C 180,E1 -4359.443,E2 -4359.443} C_VEL
LIN {X 0,Y 530.981,Z 51.345,A -85,B 0,C 180,E1 -4362.457,E2 -4362.457} C_VEL
LIN {X 0,Y 530.979,Z 51.339,A -85,B 0,C 180,E1 -4365.622,E2 -4365.622} C_VEL
LIN {X 0,Y 530.996,Z 51.344,A -85,B 0,C 180,E1 -4368.564,E2 -4368.564} C_VEL
LIN {X 0,Y 530.96,Z 51.342,A -85,B 0,C 180,E1 -4371.529,E2 -4371.529} C_VEL
LIN {X 0,Y 530.957,Z 51.347,A -85,B 0,C 180,E1 -4374.38,E2 -4374.38} C_VEL
LIN {X 0,Y 530.97,Z 51.343,A -85,B 0,C 180,E1 -4377.133,E2 -4377.133} C_VEL
LIN {X 0,Y 530.972,Z 51.348,A -85,B 0,C 180,E1 -4379.803,E2 -4379.803} C_VEL
LIN {X 0,Y 531.017,Z 51.339,A -85,B 0,C 180,E1 -4382.467,E2 -4382.467} C_VEL
LIN {X 0,Y 531.064,Z 51.502,A -85,B 0,C 180,E1 -4385.259,E2 -4385.259} C_VEL
LIN {X 0,Y 532.308,Z 58.942,A -85,B 0,C 180,E1 -4386.46,E2 -4386.46} C_VEL
LIN {X 0,Y 532.053,Z 72.414,A -85,B 0,C 180,E1 -4388.496,E2 -4388.496} C_VEL
LIN {X 0,Y 531.686,Z 89.942,A -85,B 0,C 180,E1 -4391.104,E2 -4391.104} C_VEL
LIN {X 0,Y 531.345,Z 108.809,A -85,B 0,C 180,E1 -4393.873,E2 -4393.873} C_VEL
LIN {X 0,Y 531.2,Z 116.799,A -85,B 0,C 180,E1 -4395.037,E2 -4395.037} C_VEL
LIN {X 0,Y 532.73,Z 128.647,A -85,B 0,C 180,E1 -4395.246,E2 -4395.246} C_VEL
LIN {X 0,Y 532.381,Z 225.316,A -85,B 0,C 180,E1 -4396.57,E2 -4396.57} C_VEL
LIN {X 0,Y 532.157,Z 238.638,A -85,B 0,C 180,E1 -4396.904,E2 -4396.904} C_VEL
LIN {X 0,Y 531.93,Z 251.968,A -85,B 0,C 180,E1 -4397.408,E2 -4397.408} C_VEL
LIN {X 0,Y 531.661,Z 264.537,A -85,B 0,C 180,E1 -4398.067,E2 -4398.067} C_VEL
LIN {X 0,Y 531.406,Z 276.088,A -85,B 0,C 180,E1 -4398.847,E2 -4398.847} C_VEL
LIN {X 0,Y 531.134,Z 286.316,A -85,B 0,C 180,E1 -4399.71,E2 -4399.71} C_VEL
LIN {X 0,Y 530.938,Z 295.523,A -85,B 0,C 180,E1 -4400.668,E2 -4400.668} C_VEL
LIN {X 0,Y 530.742,Z 304.496,A -85,B 0,C 180,E1 -4401.816,E2 -4401.816} C_VEL
LIN {X 0,Y 530.587,Z 311.719,A -85,B 0,C 180,E1 -4402.962,E2 -4402.962} C_VEL
LIN {X 0,Y 530.563,Z 318.303,A -85,B 0,C 180,E1 -4404.298,E2 -4404.298} C_VEL
LIN {X 0,Y 530.449,Z 322.655,A -85,B 0,C 180,E1 -4405.44,E2 -4405.44} C_VEL
LIN {X 0,Y 530.516,Z 324.964,A -85,B 0,C 180,E1 -4406.202,E2 -4406.202} C_VEL
LIN {X 0,Y 530.483,Z 326.833,A -85,B 0,C 180,E1 -4406.962,E2 -4406.962} C_VEL
LIN {X 0,Y 530.412,Z 328.231,A -85,B 0,C 180,E1 -4407.722,E2 -4407.722} C_VEL
LIN {X 0,Y 530.361,Z 329.842,A -85,B 0,C 180,E1 -4409.241,E2 -4409.241} C_VEL
LIN {X 0,Y 530.363,Z 330.06,A -85,B 0,C 180,E1 -4410,E2 -4410} C_VEL
LIN {X 0,Y 530.361,Z 329.844,A -85,B 0,C 180,E1 -4410.759,E2 -4410.759} C_VEL
LIN {X 0,Y 530.412,Z 328.241,A -85,B 0,C 180,E1 -4412.278,E2 -4412.278} C_VEL
LIN {X 0,Y 530.482,Z 326.844,A -85,B 0,C 180,E1 -4413.037,E2 -4413.037} C_VEL
LIN {X 0,Y 530.52,Z 323.901,A -85,B 0,C 180,E1 -4414.178,E2 -4414.178} C_VEL
LIN {X 0,Y 530.52,Z 319.915,A -85,B 0,C 180,E1 -4415.321,E2 -4415.321} C_VEL
LIN {X 0,Y 530.54,Z 314.469,A -85,B 0,C 180,E1 -4416.527,E2 -4416.527} C_VEL
LIN {X 0,Y 530.673,Z 308.329,A -85,B 0,C 180,E1 -4417.61,E2 -4417.61} C_VEL
LIN {X 0,Y 530.823,Z 300.277,A -85,B 0,C 180,E1 -4418.758,E2 -4418.758} C_VEL
LIN {X 0,Y 531.001,Z 292.073,A -85,B 0,C 180,E1 -4419.715,E2 -4419.715} C_VEL
LIN {X 0,Y 531.28,Z 282.075,A -85,B 0,C 180,E1 -4420.672,E2 -4420.672} C_VEL
LIN {X 0,Y 531.491,Z 270.675,A -85,B 0,C 180,E1 -4421.544,E2 -4421.544} C_VEL
LIN {X 0,Y 531.781,Z 259.731,A -85,B 0,C 180,E1 -4422.207,E2 -4422.207} C_VEL
LIN {X 0,Y 532.024,Z 247.483,A -85,B 0,C 180,E1 -4422.783,E2 -4422.783} C_VEL
LIN {X 0,Y 532.233,Z 234.632,A -85,B 0,C 180,E1 -4423.215,E2 -4423.215} C_VEL
LIN {X 0,Y 532.459,Z 221.013,A -85,B 0,C 180,E1 -4423.501,E2 -4423.501} C_VEL
LIN {X 0,Y 532.619,Z 126.524,A -85,B 0,C 180,E1 -4424.787,E2 -4424.787} C_VEL
LIN {X 0,Y 531.21,Z 116.824,A -85,B 0,C 180,E1 -4424.966,E2 -4424.966} C_VEL
LIN {X 0,Y 531.57,Z 98.095,A -85,B 0,C 180,E1 -4427.703,E2 -4427.703} C_VEL
LIN {X 0,Y 531.995,Z 76.521,A -85,B 0,C 180,E1 -4430.897,E2 -4430.897} C_VEL
LIN {X 0,Y 532.33,Z 60.278,A -85,B 0,C 180,E1 -4433.333,E2 -4433.333} C_VEL
LIN {X 0,Y 531.707,Z 54.807,A -85,B 0,C 180,E1 -4434.189,E2 -4434.189} C_VEL
LIN {X 0,Y 531.055,Z 51.336,A -85,B 0,C 180,E1 -4434.767,E2 -4434.767} C_VEL
LIN {X 0,Y 531.017,Z 51.339,A -85,B 0,C 180,E1 -4437.595,E2 -4437.595} C_VEL
LIN {X 0,Y 530.975,Z 51.34,A -85,B 0,C 180,E1 -4440.645,E2 -4440.645} C_VEL
LIN {X 0,Y 530.988,Z 51.346,A -85,B 0,C 180,E1 -4443.772,E2 -4443.772} C_VEL
LIN {X 0,Y 530.956,Z 51.342,A -85,B 0,C 180,E1 -4446.558,E2 -4446.558} C_VEL
LIN {X 0,Y 530.99,Z 51.343,A -85,B 0,C 180,E1 -4449.443,E2 -4449.443} C_VEL
LIN {X 0,Y 530.978,Z 51.339,A -85,B 0,C 180,E1 -4452.457,E2 -4452.457} C_VEL
LIN {X 0,Y 530.976,Z 51.346,A -85,B 0,C 180,E1 -4455.622,E2 -4455.622} C_VEL
LIN {X 0,Y 530.993,Z 51.337,A -85,B 0,C 180,E1 -4458.564,E2 -4458.564} C_VEL
LIN {X 0,Y 530.955,Z 51.348,A -85,B 0,C 180,E1 -4461.529,E2 -4461.529} C_VEL
LIN {X 0,Y 530.958,Z 51.342,A -85,B 0,C 180,E1 -4464.38,E2 -4464.38} C_VEL
LIN {X 0,Y 530.967,Z 51.35,A -85,B 0,C 180,E1 -4467.133,E2 -4467.133} C_VEL
LIN {X 0,Y 530.969,Z 51.341,A -85,B 0,C 180,E1 -4469.803,E2 -4469.803} C_VEL
LIN {X 0,Y 531.012,Z 51.337,A -85,B 0,C 180,E1 -4472.467,E2 -4472.467} C_VEL
LIN {X 0,Y 530.995,Z 51.345,A -85,B 0,C 180,E1 -4474.942,E2 -4474.942} C_VEL
LIN {X 0,Y 530.971,Z 51.342,A -85,B 0,C 180,E1 -4478.247,E2 -4478.247} C_VEL
LIN {X 0,Y 530.992,Z 51.346,A -85,B 0,C 180,E1 -4480.677,E2 -4480.677} C_VEL
LIN {X 0,Y 530.969,Z 51.343,A -85,B 0,C 180,E1 -4483.071,E2 -4483.071} C_VEL
LIN {X 0,Y 531.016,Z 51.334,A -85,B 0,C 180,E1 -4485.436,E2 -4485.436} C_VEL
LIN {X 0,Y 531.035,Z 51.34,A -85,B 0,C 180,E1 -4488.55,E2 -4488.55} C_VEL
LIN {X 0,Y 531.051,Z 51.331,A -85,B 0,C 180,E1 -4491.63,E2 -4491.63} C_VEL
LIN {X 0,Y 531.116,Z 51.325,A -85,B 0,C 180,E1 -4494.685,E2 -4494.685} C_VEL
LIN {X 0,Y 531.14,Z 51.322,A -85,B 0,C 180,E1 -4497.725,E2 -4497.725} C_VEL
LIN {X 0,Y 531.148,Z 51.319,A -85,B 0,C 180,E1 -4500.758,E2 -4500.758} C_VEL
LIN {X 0,Y 531.1,Z 51.324,A -85,B 0,C 180,E1 -4503.034,E2 -4503.034} C_VEL
LIN {X 0,Y 531.069,Z 51.334,A -85,B 0,C 180,E1 -4506.077,E2 -4506.077} C_VEL
LIN {X 0,Y 531.016,Z 51.335,A -85,B 0,C 180,E1 -4509.139,E2 -4509.139} C_VEL
LIN {X 0,Y 531.05,Z 51.339,A -85,B 0,C 180,E1 -4511.671,E2 -4511.671} C_VEL
LIN {X 0,Y 531.029,Z 51.334,A -85,B 0,C 180,E1 -4514.955,E2 -4514.955} C_VEL
LIN {X 0,Y 530.98,Z 51.345,A -85,B 0,C 180,E1 -4517.724,E2 -4517.724} C_VEL
LIN {X 0,Y 531.025,Z 51.334,A -85,B 0,C 180,E1 -4520.127,E2 -4520.127} C_VEL
LIN {X 0,Y 530.942,Z 51.344,A -85,B 0,C 180,E1 -4522.574,E2 -4522.574} C_VEL
LIN {X 0,Y 530.966,Z 51.346,A -85,B 0,C 180,E1 -4525.06,E2 -4525.06} C_VEL
LIN {X 0,Y 531.011,Z 51.339,A -85,B 0,C 180,E1 -4527.596,E2 -4527.596} C_VEL
LIN {X 0,Y 530.966,Z 51.343,A -85,B 0,C 180,E1 -4530.644,E2 -4530.644} C_VEL
LIN {X 0,Y 530.963,Z 51.344,A -85,B 0,C 180,E1 -4533.5,E2 -4533.5} C_VEL
LIN {X 0,Y 530.956,Z 51.345,A -85,B 0,C 180,E1 -4536.559,E2 -4536.559} C_VEL
LIN {X 0,Y 530.971,Z 51.341,A -85,B 0,C 180,E1 -4539.445,E2 -4539.445} C_VEL
LIN {X 0,Y 530.932,Z 51.349,A -85,B 0,C 180,E1 -4542.462,E2 -4542.462} C_VEL
LIN {X 0,Y 530.938,Z 51.344,A -85,B 0,C 180,E1 -4543.538,E2 -4543.538} C_VEL
LIN {X 0,Y 530.268,Z 51.43,A -85,B 0,C 180,E1 -4544.172,E2 -4544.172} C_VEL
LIN {X 0,Y 527.423,Z 51.79,A -85,B 0,C 180,E1 -4545.201,E2 -4545.201} C_VEL
LIN {X 0,Y 525.019,Z 52.092,A -85,B 0,C 180,E1 -4546.029,E2 -4546.029} C_VEL
LIN {X 0,Y 523.986,Z 52.218,A -85,B 0,C 180,E1 -4546.669,E2 -4546.669} C_VEL
LIN {X 0,Y 523.902,Z 52.225,A -85,B 0,C 180,E1 -4546.885,E2 -4546.885} C_VEL
LIN {X 0,Y 523.936,Z 52.218,A -85,B 0,C 180,E1 -4549.92,E2 -4549.92} C_VEL
LIN {X 0,Y 523.899,Z 52.224,A -85,B 0,C 180,E1 -4552.867,E2 -4552.867} C_VEL
LIN {X 0,Y 523.928,Z 52.219,A -85,B 0,C 180,E1 -4555.71,E2 -4555.71} C_VEL
LIN {X 0,Y 523.924,Z 52.224,A -85,B 0,C 180,E1 -4558.456,E2 -4558.456} C_VEL
LIN {X 0,Y 523.929,Z 52.217,A -85,B 0,C 180,E1 -4561.125,E2 -4561.125} C_VEL
LIN {X 0,Y 523.912,Z 52.227,A -85,B 0,C 180,E1 -4563.998,E2 -4563.998} C_VEL
LIN {X 0,Y 523.913,Z 52.224,A -85,B 0,C 180,E1 -4566.27,E2 -4566.27} C_VEL
LIN {X 0,Y 523.949,Z 52.215,A -85,B 0,C 180,E1 -4568.767,E2 -4568.767} C_VEL
LIN {X 0,Y 523.939,Z 52.217,A -85,B 0,C 180,E1 -4571.22,E2 -4571.22} C_VEL
LIN {X 0,Y 523.917,Z 52.226,A -85,B 0,C 180,E1 -4573.638,E2 -4573.638} C_VEL
LIN {X 0,Y 523.928,Z 52.225,A -85,B 0,C 180,E1 -4576.028,E2 -4576.028} C_VEL
LIN {X 0,Y 524.001,Z 52.234,A -85,B 0,C 180,E1 -4577.843,E2 -4577.843} C_VEL
LIN {X 0,Y 524.496,Z 56.885,A -85,B 0,C 180,E1 -4578.797,E2 -4578.797} C_VEL
LIN {X 0,Y 524.4,Z 68.61,A -85,B 0,C 180,E1 -4581.134,E2 -4581.134} C_VEL
LIN {X 0,Y 524.275,Z 72.545,A -85,B 0,C 180,E1 -4581.908,E2 -4581.908} C_VEL
LIN {X 0,Y 525.984,Z 81.387,A -85,B 0,C 180,E1 -4582.083,E2 -4582.083} C_VEL
LIN {X 0,Y 525.502,Z 179.435,A -85,B 0,C 180,E1 -4583.449,E2 -4583.449} C_VEL
LIN {X 0,Y 525.326,Z 193.099,A -85,B 0,C 180,E1 -4583.808,E2 -4583.808} C_VEL
LIN {X 0,Y 525.195,Z 205.347,A -85,B 0,C 180,E1 -4584.288,E2 -4584.288} C_VEL
LIN {X 0,Y 525.001,Z 217.101,A -85,B 0,C 180,E1 -4584.912,E2 -4584.912} C_VEL
LIN {X 0,Y 524.688,Z 228.39,A -85,B 0,C 180,E1 -4585.679,E2 -4585.679} C_VEL
LIN {X 0,Y 524.392,Z 238.581,A -85,B 0,C 180,E1 -4586.543,E2 -4586.543} C_VEL
LIN {X 0,Y 524.157,Z 247.765,A -85,B 0,C 180,E1 -4587.503,E2 -4587.503} C_VEL
LIN {X 0,Y 523.857,Z 256.671,A -85,B 0,C 180,E1 -4588.655,E2 -4588.655} C_VEL
LIN {X 0,Y 523.752,Z 263.85,A -85,B 0,C 180,E1 -4589.808,E2 -4589.808} C_VEL
LIN {X 0,Y 523.52,Z 270.463,A -85,B 0,C 180,E1 -4591.154,E2 -4591.154} C_VEL
LIN {X 0,Y 523.418,Z 274.838,A -85,B 0,C 180,E1 -4592.309,E2 -4592.309} C_VEL
LIN {X 0,Y 523.456,Z 277.146,A -85,B 0,C 180,E1 -4593.079,E2 -4593.079} C_VEL
LIN {X 0,Y 523.409,Z 279.042,A -85,B 0,C 180,E1 -4593.85,E2 -4593.85} C_VEL
LIN {X 0,Y 523.336,Z 280.513,A -85,B 0,C 180,E1 -4594.622,E2 -4594.622} C_VEL
LIN {X 0,Y 523.401,Z 282.185,A -85,B 0,C 180,E1 -4596.167,E2 -4596.167} C_VEL
LIN {X 0,Y 523.371,Z 282.452,A -85,B 0,C 180,E1 -4596.942,E2 -4596.942} C_VEL
LIN {X 0,Y 523.362,Z 282.316,A -85,B 0,C 180,E1 -4597.718,E2 -4597.718} C_VEL
LIN {X 0,Y 523.361,Z 281.752,A -85,B 0,C 180,E1 -4598.495,E2 -4598.495} C_VEL
LIN {X 0,Y 523.366,Z 279.448,A -85,B 0,C 180,E1 -4600.054,E2 -4600.054} C_VEL
LIN {X 0,Y 523.443,Z 275.948,A -85,B 0,C 180,E1 -4601.437,E2 -4601.437} C_VEL
LIN {X 0,Y 523.529,Z 271.058,A -85,B 0,C 180,E1 -4602.797,E2 -4602.797} C_VEL
LIN {X 0,Y 523.712,Z 265.514,A -85,B 0,C 180,E1 -4603.978,E2 -4603.978} C_VEL
LIN {X 0,Y 523.847,Z 258.504,A -85,B 0,C 180,E1 -4605.172,E2 -4605.172} C_VEL
LIN {X 0,Y 524.073,Z 249.726,A -85,B 0,C 180,E1 -4606.357,E2 -4606.357} C_VEL
LIN {X 0,Y 524.335,Z 240.73,A -85,B 0,C 180,E1 -4607.341,E2 -4607.341} C_VEL
LIN {X 0,Y 524.549,Z 230.545,A -85,B 0,C 180,E1 -4608.251,E2 -4608.251} C_VEL
LIN {X 0,Y 524.851,Z 219.255,A -85,B 0,C 180,E1 -4609.05,E2 -4609.05} C_VEL
LIN {X 0,Y 525.153,Z 206.497,A -85,B 0,C 180,E1 -4609.75,E2 -4609.75} C_VEL
LIN {X 0,Y 525.381,Z 194.069,A -85,B 0,C 180,E1 -4610.251,E2 -4610.251} C_VEL
LIN {X 0,Y 525.541,Z 181.725,A -85,B 0,C 180,E1 -4610.592,E2 -4610.592} C_VEL
LIN {X 0,Y 525.635,Z 162.821,A -85,B 0,C 180,E1 -4610.89,E2 -4610.89} C_VEL
LIN {X 0,Y 525.869,Z 80.479,A -85,B 0,C 180,E1 -4612.024,E2 -4612.024} C_VEL
LIN {X 0,Y 524.332,Z 72.526,A -85,B 0,C 180,E1 -4612.196,E2 -4612.196} C_VEL
LIN {X 0,Y 524.56,Z 57.558,A -85,B 0,C 180,E1 -4615.175,E2 -4615.175} C_VEL
LIN {X 0,Y 523.952,Z 52.223,A -85,B 0,C 180,E1 -4616.3,E2 -4616.3} C_VEL
LIN {X 0,Y 523.939,Z 52.219,A -85,B 0,C 180,E1 -4619.319,E2 -4619.319} C_VEL
LIN {X 0,Y 523.9,Z 52.228,A -85,B 0,C 180,E1 -4622.452,E2 -4622.452} C_VEL
LIN {X 0,Y 523.886,Z 52.224,A -85,B 0,C 180,E1 -4625.23,E2 -4625.23} C_VEL
LIN {X 0,Y 523.892,Z 52.23,A -85,B 0,C 180,E1 -4628.104,E2 -4628.104} C_VEL
LIN {X 0,Y 523.879,Z 52.226,A -85,B 0,C 180,E1 -4631.3,E2 -4631.3} C_VEL
LIN {X 0,Y 523.934,Z 52.212,A -85,B 0,C 180,E1 -4634.688,E2 -4634.688} C_VEL
LIN {X 0,Y 523.891,Z 52.227,A -85,B 0,C 180,E1 -4637.874,E2 -4637.874} C_VEL
LIN {X 0,Y 523.886,Z 52.226,A -85,B 0,C 180,E1 -4641.085,E2 -4641.085} C_VEL
LIN {X 0,Y 523.854,Z 52.23,A -85,B 0,C 180,E1 -4643.821,E2 -4643.821} C_VEL
LIN {X 0,Y 523.899,Z 52.222,A -85,B 0,C 180,E1 -4646.632,E2 -4646.632} C_VEL
LIN {X 0,Y 523.91,Z 52.228,A -85,B 0,C 180,E1 -4649.352,E2 -4649.352} C_VEL
LIN {X 0,Y 523.915,Z 52.218,A -85,B 0,C 180,E1 -4652.295,E2 -4652.295} C_VEL
LIN {X 0,Y 523.896,Z 52.225,A -85,B 0,C 180,E1 -4655.426,E2 -4655.426} C_VEL
LIN {X 0,Y 523.94,Z 52.214,A -85,B 0,C 180,E1 -4657.939,E2 -4657.939} C_VEL
LIN {X 0,Y 523.96,Z 52.216,A -85,B 0,C 180,E1 -4660.407,E2 -4660.407} C_VEL
LIN {X 0,Y 523.942,Z 52.221,A -85,B 0,C 180,E1 -4662.836,E2 -4662.836} C_VEL
LIN {X 0,Y 523.964,Z 52.215,A -85,B 0,C 180,E1 -4665.235,E2 -4665.235} C_VEL
LIN {X 0,Y 524.017,Z 52.209,A -85,B 0,C 180,E1 -4668.394,E2 -4668.394} C_VEL
LIN {X 0,Y 523.962,Z 52.213,A -85,B 0,C 180,E1 -4671.515,E2 -4671.515} C_VEL
LIN {X 0,Y 524.033,Z 52.209,A -85,B 0,C 180,E1 -4674.613,E2 -4674.613} C_VEL
LIN {X 0,Y 524.106,Z 52.197,A -85,B 0,C 180,E1 -4677.694,E2 -4677.694} C_VEL
LIN {X 0,Y 524.121,Z 52.193,A -85,B 0,C 180,E1 -4680.768,E2 -4680.768} C_VEL
LIN {X 0,Y 524.005,Z 52.208,A -85,B 0,C 180,E1 -4683.075,E2 -4683.075} C_VEL
LIN {X 0,Y 524.011,Z 52.211,A -85,B 0,C 180,E1 -4686.159,E2 -4686.159} C_VEL
LIN {X 0,Y 523.984,Z 52.212,A -85,B 0,C 180,E1 -4689.262,E2 -4689.262} C_VEL
LIN {X 0,Y 524.002,Z 52.212,A -85,B 0,C 180,E1 -4691.737,E2 -4691.737} C_VEL
LIN {X 0,Y 523.99,Z 52.211,A -85,B 0,C 180,E1 -4695.049,E2 -4695.049} C_VEL
LIN {X 0,Y 523.919,Z 52.221,A -85,B 0,C 180,E1 -4697.971,E2 -4697.971} C_VEL
LIN {X 0,Y 523.961,Z 52.213,A -85,B 0,C 180,E1 -4700.41,E2 -4700.41} C_VEL
LIN {X 0,Y 523.911,Z 52.219,A -85,B 0,C 180,E1 -4702.894,E2 -4702.894} C_VEL
LIN {X 0,Y 523.912,Z 52.225,A -85,B 0,C 180,E1 -4705.421,E2 -4705.421} C_VEL
LIN {X 0,Y 523.959,Z 52.214,A -85,B 0,C 180,E1 -4708,E2 -4708} C_VEL
LIN {X 0,Y 523.938,Z 52.221,A -85,B 0,C 180,E1 -4710.853,E2 -4710.853} C_VEL
LIN {X 0,Y 523.963,Z 52.213,A -85,B 0,C 180,E1 -4713.734,E2 -4713.734} C_VEL
LIN {X 0,Y 523.906,Z 52.217,A -85,B 0,C 180,E1 -4716.401,E2 -4716.401} C_VEL
LIN {X 0,Y 523.921,Z 52.223,A -85,B 0,C 180,E1 -4719.085,E2 -4719.085} C_VEL
LIN {X 0,Y 523.954,Z 52.216,A -85,B 0,C 180,E1 -4722.119,E2 -4722.119} C_VEL
LIN {X 0,Y 523.945,Z 52.216,A -85,B 0,C 180,E1 -4725.31,E2 -4725.31} C_VEL
LIN {X 0,Y 523.959,Z 52.219,A -85,B 0,C 180,E1 -4728.69,E2 -4728.69} C_VEL
LIN {X 0,Y 523.921,Z 52.219,A -85,B 0,C 180,E1 -4731.08,E2 -4731.08} C_VEL
LIN {X 0,Y 523.903,Z 52.224,A -85,B 0,C 180,E1 -4733.825,E2 -4733.825} C_VEL
LIN {X 0,Y 523.944,Z 52.221,A -85,B 0,C 180,E1 -4736.635,E2 -4736.635} C_VEL
LIN {X 0,Y 523.959,Z 52.218,A -85,B 0,C 180,E1 -4739.356,E2 -4739.356} C_VEL
LIN {X 0,Y 523.979,Z 52.218,A -85,B 0,C 180,E1 -4742.282,E2 -4742.282} C_VEL
LIN {X 0,Y 524.008,Z 52.309,A -85,B 0,C 180,E1 -4745.062,E2 -4745.062} C_VEL
LIN {X 0,Y 525.371,Z 60.069,A -85,B 0,C 180,E1 -4746.339,E2 -4746.339} C_VEL
LIN {X 0,Y 525.09,Z 73.51,A -85,B 0,C 180,E1 -4748.403,E2 -4748.403} C_VEL
LIN {X 0,Y 524.691,Z 90.992,A -85,B 0,C 180,E1 -4751.045,E2 -4751.045} C_VEL
LIN {X 0,Y 524.369,Z 108.488,A -85,B 0,C 180,E1 -4753.652,E2 -4753.652} C_VEL
LIN {X 0,Y 524.18,Z 116.394,A -85,B 0,C 180,E1 -4754.82,E2 -4754.82} C_VEL
LIN {X 0,Y 525.86,Z 128.445,A -85,B 0,C 180,E1 -4755.05,E2 -4755.05} C_VEL
LIN {X 0,Y 525.471,Z 224.974,A -85,B 0,C 180,E1 -4756.39,E2 -4756.39} C_VEL
LIN {X 0,Y 525.248,Z 238.302,A -85,B 0,C 180,E1 -4756.729,E2 -4756.729} C_VEL
LIN {X 0,Y 524.964,Z 251.633,A -85,B 0,C 180,E1 -4757.238,E2 -4757.238} C_VEL
LIN {X 0,Y 524.71,Z 264.04,A -85,B 0,C 180,E1 -4757.896,E2 -4757.896} C_VEL
LIN {X 0,Y 524.417,Z 275.758,A -85,B 0,C 180,E1 -4758.697,E2 -4758.697} C_VEL
LIN {X 0,Y 524.142,Z 285.988,A -85,B 0,C 180,E1 -4759.571,E2 -4759.571} C_VEL
LIN {X 0,Y 523.896,Z 295.194,A -85,B 0,C 180,E1 -4760.541,E2 -4760.541} C_VEL
LIN {X 0,Y 523.666,Z 304.168,A -85,B 0,C 180,E1 -4761.705,E2 -4761.705} C_VEL
LIN {X 0,Y 523.513,Z 311.393,A -85,B 0,C 180,E1 -4762.866,E2 -4762.866} C_VEL
LIN {X 0,Y 523.474,Z 317.978,A -85,B 0,C 180,E1 -4764.221,E2 -4764.221} C_VEL
LIN {X 0,Y 523.354,Z 322.331,A -85,B 0,C 180,E1 -4765.378,E2 -4765.378} C_VEL
LIN {X 0,Y 523.443,Z 324.642,A -85,B 0,C 180,E1 -4766.15,E2 -4766.15} C_VEL
LIN {X 0,Y 523.391,Z 326.51,A -85,B 0,C 180,E1 -4766.921,E2 -4766.921} C_VEL
LIN {X 0,Y 523.337,Z 327.911,A -85,B 0,C 180,E1 -4767.691,E2 -4767.691} C_VEL
LIN {X 0,Y 523.268,Z 329.521,A -85,B 0,C 180,E1 -4769.23,E2 -4769.23} C_VEL
LIN {X 0,Y 523.271,Z 329.74,A -85,B 0,C 180,E1 -4770,E2 -4770} C_VEL
LIN {X 0,Y 523.279,Z 328.916,A -85,B 0,C 180,E1 -4771.539,E2 -4771.539} C_VEL
LIN {X 0,Y 523.337,Z 327.922,A -85,B 0,C 180,E1 -4772.309,E2 -4772.309} C_VEL
LIN {X 0,Y 523.39,Z 326.524,A -85,B 0,C 180,E1 -4773.079,E2 -4773.079} C_VEL
LIN {X 0,Y 523.421,Z 323.581,A -85,B 0,C 180,E1 -4774.235,E2 -4774.235} C_VEL
LIN {X 0,Y 523.453,Z 319.595,A -85,B 0,C 180,E1 -4775.393,E2 -4775.393} C_VEL
LIN {X 0,Y 523.49,Z 313.553,A -85,B 0,C 180,E1 -4776.729,E2 -4776.729} C_VEL
LIN {X 0,Y 523.64,Z 306.768,A -85,B 0,C 180,E1 -4777.907,E2 -4777.907} C_VEL
LIN {X 0,Y 523.806,Z 298.459,A -85,B 0,C 180,E1 -4779.07,E2 -4779.07} C_VEL
LIN {X 0,Y 523.985,Z 289.945,A -85,B 0,C 180,E1 -4780.041,E2 -4780.041} C_VEL
LIN {X 0,Y 524.285,Z 279.43,A -85,B 0,C 180,E1 -4781.012,E2 -4781.012} C_VEL
LIN {X 0,Y 524.62,Z 267.699,A -85,B 0,C 180,E1 -4781.879,E2 -4781.879} C_VEL
LIN {X 0,Y 524.912,Z 255.704,A -85,B 0,C 180,E1 -4782.566,E2 -4782.566} C_VEL
LIN {X 0,Y 525.134,Z 243.332,A -85,B 0,C 180,E1 -4783.101,E2 -4783.101} C_VEL
